KUKA KRL program: EPS_2_26115_ST7264_A_20260223020928.src

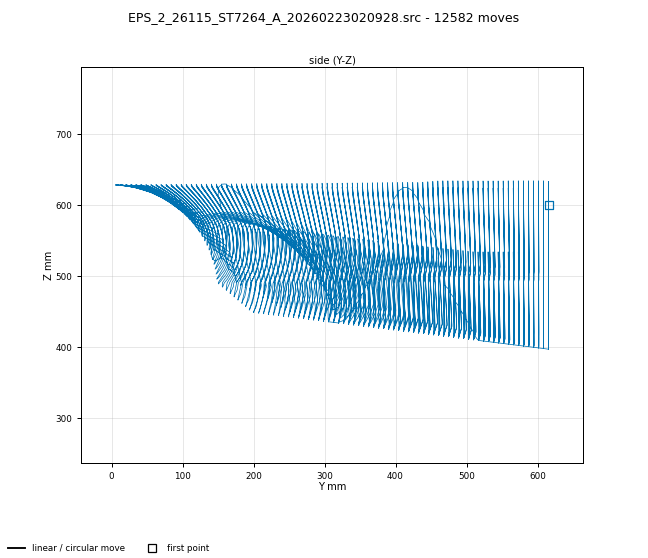
[picture p0: tool path of EPS_2_26115_ST7264_A_20260223020928.src, 12582 of 12584 moves have a stored position in this frame; points joined in program order, loops and branches not executed]
&ACCESS RVP
&REL 4
&COMMENT QRS 19112012
&PARAM EDITMASK = *
DEF PART()
EXT BAS (BAS_COMMAND :IN,REAL :IN )
INT I
BAS (#INITMOV,0 )

;KUKA QRS Post kuka4.cps  Date:22-06-2017 !

File_ID=3073

QRS_PRE_INIT()

;Init var - Until changes are made in qrs_pre_init
Outlet_Square_prg=0
Inlet_1_Square_prg=0
Inlet_2_Square_prg=0
Inlet_3_Square_prg=0
Inlet_4_Square_prg=0
Inlet_5_Square_prg=0

Outlet_1={X 0.000, Y 460.000, Z 509.000, B 0.000, E1 0.000 }
Inlet_1={X 0.000, Y 510.210, Z 499.000, B 0.000, E1 180.000 }
Inlet_2={X 0.000, Y 509.920, Z 385.000, B 0.000, E1 270.000 }
Outlet_1_type=251
Inlet_1_type=251
Inlet_2_type=299
;QRS#1=Sidecore dimensions
;QRS#2=250-10" PVC SDR 35 Cut Back
;QRS#3=250-10" PVC SDR 35
;QRS#4=300-12" PVC SDR 35
;QRS#5=
;QRS#6=
;QRS#7=
;QRS#8=
;QRS#9=14M PSX
;QRS#10=14M PSX
;QRS#11=16M PSX
;QRS#12=
;QRS#13=
;QRS#14=
;QRS#15=
;QRS#16=1220x127x914 3'
;QRS#17=EPS Height
;QRS#18=634,5
;QRS#19=*
;QRS#20= UPDATED VERSION 22-06-2017
;QRS#21=*
Outlet_Square=0100
Inlet_1_Square=0100
Inlet_2_Square=0150
Inlet_3_Square=0
Inlet_4_Square=0
Inlet_5_Square=0
Mill_Square=1
Outlet_Square_Prg=215
Inlet_1_Square_prg=205
Inlet_2_Square_prg=206

QRS_INIT()

$ADVANCE=5

; T1
PTP {E1 173.607,E2 173.607}
PTP {X 0,Y 615.507,A -85,B 0,C 180,E1 173.607,E2 173.607,E3 0,E4 0,E5 0,E6 0}
QRS_SPEED_INIT()
LIN {X 0,Y 615.507,Z 600,A -85,B 0,C 180,E1 173.607,E2 173.607,E3 0,E4 0,E5 0,E6 0} C_VEL
LIN {X 0,Y 615.507,Z 407.495,A -85,B 0,C 180,E1 173.607,E2 173.607} C_VEL
LIN {X 0,Y 615.507,Z 399.316,A -85,B 0,C 180,E1 173.607,E2 173.607} C_VEL
LIN {X 0,Y 615.491,Z 397.316,A -85,B 0,C 180,E1 173.42,E2 173.42} C_VEL
LIN {X 0,Y 615.489,Z 397.323,A -85,B 0,C 180,E1 170.801,E2 170.801} C_VEL
LIN {X 0,Y 615.489,Z 397.323,A -85,B 0,C 180,E1 168.139,E2 168.139} C_VEL
LIN {X 0,Y 615.493,Z 397.316,A -85,B 0,C 180,E1 165.451,E2 165.451} C_VEL
LIN {X 0,Y 615.49,Z 397.315,A -85,B 0,C 180,E1 162.729,E2 162.729} C_VEL
LIN {X 0,Y 615.484,Z 397.318,A -85,B 0,C 180,E1 159.967,E2 159.967} C_VEL
LIN {X 0,Y 615.477,Z 397.323,A -85,B 0,C 180,E1 157.155,E2 157.155} C_VEL
LIN {X 0,Y 615.499,Z 397.325,A -85,B 0,C 180,E1 154.429,E2 154.429} C_VEL
LIN {X 0,Y 615.497,Z 397.322,A -85,B 0,C 180,E1 151.548,E2 151.548} C_VEL
LIN {X 0,Y 615.483,Z 397.318,A -85,B 0,C 180,E1 148.915,E2 148.915} C_VEL
LIN {X 0,Y 615.484,Z 397.319,A -85,B 0,C 180,E1 146.466,E2 146.466} C_VEL
LIN {X 0,Y 615.488,Z 397.32,A -85,B 0,C 180,E1 143.575,E2 143.575} C_VEL
LIN {X 0,Y 615.496,Z 397.324,A -85,B 0,C 180,E1 140.937,E2 140.937} C_VEL
LIN {X 0,Y 615.485,Z 397.317,A -85,B 0,C 180,E1 138.526,E2 138.526} C_VEL
LIN {X 0,Y 615.495,Z 397.315,A -85,B 0,C 180,E1 135.851,E2 135.851} C_VEL
LIN {X 0,Y 615.485,Z 397.321,A -85,B 0,C 180,E1 133.047,E2 133.047} C_VEL
LIN {X 0,Y 615.492,Z 397.32,A -85,B 0,C 180,E1 130.089,E2 130.089} C_VEL
LIN {X 0,Y 615.497,Z 397.512,A -85,B 0,C 180,E1 127.721,E2 127.721} C_VEL
LIN {X 0,Y 615.499,Z 409.44,A -85,B 0,C 180,E1 124.814,E2 124.814} C_VEL
LIN {X 0,Y 615.489,Z 415.54,A -85,B 0,C 180,E1 123.236,E2 123.236} C_VEL
LIN {X 0,Y 615.477,Z 425.47,A -85,B 0,C 180,E1 120.54,E2 120.54} C_VEL
LIN {X 0,Y 615.485,Z 435.39,A -85,B 0,C 180,E1 117.915,E2 117.915} C_VEL
LIN {X 0,Y 615.488,Z 446.726,A -85,B 0,C 180,E1 114.992,E2 114.992} C_VEL
LIN {X 0,Y 615.49,Z 458.047,A -85,B 0,C 180,E1 112.136,E2 112.136} C_VEL
LIN {X 0,Y 615.483,Z 469.366,A -85,B 0,C 180,E1 109.338,E2 109.338} C_VEL
LIN {X 0,Y 615.48,Z 480.679,A -85,B 0,C 180,E1 106.587,E2 106.587} C_VEL
LIN {X 0,Y 615.493,Z 491.397,A -85,B 0,C 180,E1 104.013,E2 104.013} C_VEL
LIN {X 0,Y 615.494,Z 505.428,A -85,B 0,C 180,E1 103.79,E2 103.79} C_VEL
LIN {X 0,Y 615.479,Z 518.818,A -85,B 0,C 180,E1 103.454,E2 103.454} C_VEL
LIN {X 0,Y 615.493,Z 532.069,A -85,B 0,C 180,E1 102.991,E2 102.991} C_VEL
LIN {X 0,Y 615.477,Z 545.74,A -85,B 0,C 180,E1 102.363,E2 102.363} C_VEL
LIN {X 0,Y 615.499,Z 557.359,A -85,B 0,C 180,E1 101.694,E2 101.694} C_VEL
LIN {X 0,Y 615.496,Z 568.763,A -85,B 0,C 180,E1 100.891,E2 100.891} C_VEL
LIN {X 0,Y 615.498,Z 578.93,A -85,B 0,C 180,E1 100.028,E2 100.028} C_VEL
LIN {X 0,Y 615.497,Z 588.665,A -85,B 0,C 180,E1 99.033,E2 99.033} C_VEL
LIN {X 0,Y 615.498,Z 596.737,A -85,B 0,C 180,E1 98.041,E2 98.041} C_VEL
LIN {X 0,Y 615.494,Z 604.38,A -85,B 0,C 180,E1 96.899,E2 96.899} C_VEL
LIN {X 0,Y 615.497,Z 609.85,A -85,B 0,C 180,E1 95.898,E2 95.898} C_VEL
LIN {X 0,Y 615.494,Z 615.515,A -85,B 0,C 180,E1 94.585,E2 94.585} C_VEL
LIN {X 0,Y 615.494,Z 619.633,A -85,B 0,C 180,E1 93.273,E2 93.273} C_VEL
LIN {X 0,Y 615.499,Z 622.33,A -85,B 0,C 180,E1 91.963,E2 91.963} C_VEL
LIN {X 0,Y 615.491,Z 623.692,A -85,B 0,C 180,E1 90.654,E2 90.654} C_VEL
LIN {X 0,Y 615.492,Z 623.747,A -85,B 0,C 180,E1 89.346,E2 89.346} C_VEL
LIN {X 0,Y 615.499,Z 622.481,A -85,B 0,C 180,E1 88.037,E2 88.037} C_VEL
LIN {X 0,Y 615.494,Z 619.875,A -85,B 0,C 180,E1 86.727,E2 86.727} C_VEL
LIN {X 0,Y 615.495,Z 615.851,A -85,B 0,C 180,E1 85.416,E2 85.416} C_VEL
LIN {X 0,Y 615.498,Z 610.289,A -85,B 0,C 180,E1 84.102,E2 84.102} C_VEL
LIN {X 0,Y 615.495,Z 604.933,A -85,B 0,C 180,E1 83.102,E2 83.102} C_VEL
LIN {X 0,Y 615.498,Z 597.407,A -85,B 0,C 180,E1 81.959,E2 81.959} C_VEL
LIN {X 0,Y 615.496,Z 589.471,A -85,B 0,C 180,E1 80.967,E2 80.967} C_VEL
LIN {X 0,Y 615.496,Z 579.888,A -85,B 0,C 180,E1 79.972,E2 79.972} C_VEL
LIN {X 0,Y 615.497,Z 569.893,A -85,B 0,C 180,E1 79.108,E2 79.108} C_VEL
LIN {X 0,Y 615.5,Z 558.732,A -85,B 0,C 180,E1 78.306,E2 78.306} C_VEL
LIN {X 0,Y 615.48,Z 547.42,A -85,B 0,C 180,E1 77.637,E2 77.637} C_VEL
LIN {X 0,Y 615.497,Z 535.177,A -85,B 0,C 180,E1 77.051,E2 77.051} C_VEL
LIN {X 0,Y 615.48,Z 521.631,A -85,B 0,C 180,E1 76.546,E2 76.546} C_VEL
LIN {X 0,Y 615.498,Z 507.581,A -85,B 0,C 180,E1 76.168,E2 76.168} C_VEL
LIN {X 0,Y 615.489,Z 493.874,A -85,B 0,C 180,E1 75.93,E2 75.93} C_VEL
LIN {X 0,Y 615.485,Z 491.294,A -85,B 0,C 180,E1 75.872,E2 75.872} C_VEL
LIN {X 0,Y 615.491,Z 479.633,A -85,B 0,C 180,E1 73.072,E2 73.072} C_VEL
LIN {X 0,Y 615.489,Z 468.32,A -85,B 0,C 180,E1 70.315,E2 70.315} C_VEL
LIN {X 0,Y 615.487,Z 457.571,A -85,B 0,C 180,E1 67.655,E2 67.655} C_VEL
LIN {X 0,Y 615.488,Z 447.078,A -85,B 0,C 180,E1 65.008,E2 65.008} C_VEL
LIN {X 0,Y 615.485,Z 435.734,A -85,B 0,C 180,E1 62.085,E2 62.085} C_VEL
LIN {X 0,Y 615.477,Z 425.807,A -85,B 0,C 180,E1 59.46,E2 59.46} C_VEL
LIN {X 0,Y 615.492,Z 415.867,A -85,B 0,C 180,E1 56.764,E2 56.764} C_VEL
LIN {X 0,Y 615.499,Z 409.806,A -85,B 0,C 180,E1 55.186,E2 55.186} C_VEL
LIN {X 0,Y 615.496,Z 398.283,A -85,B 0,C 180,E1 52.375,E2 52.375} C_VEL
LIN {X 0,Y 615.492,Z 397.32,A -85,B 0,C 180,E1 52.085,E2 52.085} C_VEL
LIN {X 0,Y 615.482,Z 397.322,A -85,B 0,C 180,E1 49.393,E2 49.393} C_VEL
LIN {X 0,Y 615.482,Z 397.325,A -85,B 0,C 180,E1 46.755,E2 46.755} C_VEL
LIN {X 0,Y 615.486,Z 397.325,A -85,B 0,C 180,E1 43.997,E2 43.997} C_VEL
LIN {X 0,Y 615.487,Z 397.323,A -85,B 0,C 180,E1 41.474,E2 41.474} C_VEL
LIN {X 0,Y 615.476,Z 397.323,A -85,B 0,C 180,E1 38.905,E2 38.905} C_VEL
LIN {X 0,Y 615.493,Z 397.319,A -85,B 0,C 180,E1 36.425,E2 36.425} C_VEL
LIN {X 0,Y 615.486,Z 397.324,A -85,B 0,C 180,E1 33.534,E2 33.534} C_VEL
LIN {X 0,Y 615.494,Z 397.326,A -85,B 0,C 180,E1 30.919,E2 30.919} C_VEL
LIN {X 0,Y 615.497,Z 397.324,A -85,B 0,C 180,E1 28.452,E2 28.452} C_VEL
LIN {X 0,Y 615.485,Z 397.321,A -85,B 0,C 180,E1 25.568,E2 25.568} C_VEL
LIN {X 0,Y 615.481,Z 397.323,A -85,B 0,C 180,E1 22.845,E2 22.845} C_VEL
LIN {X 0,Y 615.488,Z 397.326,A -85,B 0,C 180,E1 20.033,E2 20.033} C_VEL
LIN {X 0,Y 615.49,Z 397.32,A -85,B 0,C 180,E1 17.271,E2 17.271} C_VEL
LIN {X 0,Y 615.478,Z 397.323,A -85,B 0,C 180,E1 16.037,E2 16.037} C_VEL
LIN {X 0,Y 615.485,Z 413.535,A -85,B 0,C 180,E1 15.608,E2 15.608} C_VEL
LIN {X 0,Y 615.487,Z 427.783,A -85,B 0,C 180,E1 15.099,E2 15.099} C_VEL
LIN {X 0,Y 615.496,Z 441.504,A -85,B 0,C 180,E1 14.472,E2 14.472} C_VEL
LIN {X 0,Y 615.496,Z 455.075,A -85,B 0,C 180,E1 13.706,E2 13.706} C_VEL
LIN {X 0,Y 615.496,Z 468.458,A -85,B 0,C 180,E1 12.781,E2 12.781} C_VEL
LIN {X 0,Y 615.495,Z 479.572,A -85,B 0,C 180,E1 11.861,E2 11.861} C_VEL
LIN {X 0,Y 615.493,Z 489.483,A -85,B 0,C 180,E1 10.89,E2 10.89} C_VEL
LIN {X 0,Y 615.494,Z 499.761,A -85,B 0,C 180,E1 9.696,E2 9.696} C_VEL
LIN {X 0,Y 615.496,Z 508.028,A -85,B 0,C 180,E1 8.537,E2 8.537} C_VEL
LIN {X 0,Y 615.493,Z 515.783,A -85,B 0,C 180,E1 7.216,E2 7.216} C_VEL
LIN {X 0,Y 615.489,Z 521.95,A -85,B 0,C 180,E1 5.899,E2 5.899} C_VEL
LIN {X 0,Y 615.494,Z 526.715,A -85,B 0,C 180,E1 4.585,E2 4.585} C_VEL
LIN {X 0,Y 615.495,Z 530.22,A -85,B 0,C 180,E1 3.273,E2 3.273} C_VEL
LIN {X 0,Y 615.493,Z 532.541,A -85,B 0,C 180,E1 1.963,E2 1.963} C_VEL
LIN {X 0,Y 615.489,Z 533.728,A -85,B 0,C 180,E1 0.654,E2 0.654} C_VEL
LIN {X 0,Y 615.493,Z 533.751,A -85,B 0,C 180,E1 -0.654,E2 -0.654} C_VEL
LIN {X 0,Y 615.496,Z 532.646,A -85,B 0,C 180,E1 -1.963,E2 -1.963} C_VEL
LIN {X 0,Y 615.498,Z 530.415,A -85,B 0,C 180,E1 -3.273,E2 -3.273} C_VEL
LIN {X 0,Y 615.49,Z 527.005,A -85,B 0,C 180,E1 -4.584,E2 -4.584} C_VEL
LIN {X 0,Y 615.49,Z 522.337,A -85,B 0,C 180,E1 -5.898,E2 -5.898} C_VEL
LIN {X 0,Y 615.492,Z 516.272,A -85,B 0,C 180,E1 -7.216,E2 -7.216} C_VEL
LIN {X 0,Y 615.493,Z 508.633,A -85,B 0,C 180,E1 -8.537,E2 -8.537} C_VEL
LIN {X 0,Y 615.496,Z 500.45,A -85,B 0,C 180,E1 -9.696,E2 -9.696} C_VEL
LIN {X 0,Y 615.496,Z 490.332,A -85,B 0,C 180,E1 -10.891,E2 -10.891} C_VEL
LIN {X 0,Y 615.497,Z 478.683,A -85,B 0,C 180,E1 -12.028,E2 -12.028} C_VEL
LIN {X 0,Y 615.498,Z 467.412,A -85,B 0,C 180,E1 -12.949,E2 -12.949} C_VEL
LIN {X 0,Y 615.498,Z 455.173,A -85,B 0,C 180,E1 -13.79,E2 -13.79} C_VEL
LIN {X 0,Y 615.49,Z 441.774,A -85,B 0,C 180,E1 -14.549,E2 -14.549} C_VEL
LIN {X 0,Y 615.484,Z 427.91,A -85,B 0,C 180,E1 -15.184,E2 -15.184} C_VEL
LIN {X 0,Y 615.488,Z 413.693,A -85,B 0,C 180,E1 -15.693,E2 -15.693} C_VEL
LIN {X 0,Y 615.493,Z 399.614,A -85,B 0,C 180,E1 -16.07,E2 -16.07} C_VEL
LIN {X 0,Y 615.493,Z 397.326,A -85,B 0,C 180,E1 -16.135,E2 -16.135} C_VEL
LIN {X 0,Y 615.483,Z 397.313,A -85,B 0,C 180,E1 -18.646,E2 -18.646} C_VEL
LIN {X 0,Y 615.496,Z 397.309,A -85,B 0,C 180,E1 -21.432,E2 -21.432} C_VEL
LIN {X 0,Y 615.49,Z 397.317,A -85,B 0,C 180,E1 -24.272,E2 -24.272} C_VEL
LIN {X 0,Y 615.477,Z 397.311,A -85,B 0,C 180,E1 -27.043,E2 -27.043} C_VEL
LIN {X 0,Y 615.498,Z 397.324,A -85,B 0,C 180,E1 -29.796,E2 -29.796} C_VEL
LIN {X 0,Y 615.489,Z 397.309,A -85,B 0,C 180,E1 -32.457,E2 -32.457} C_VEL
LIN {X 0,Y 615.477,Z 397.31,A -85,B 0,C 180,E1 -34.816,E2 -34.816} C_VEL
LIN {X 0,Y 615.491,Z 397.314,A -85,B 0,C 180,E1 -37.242,E2 -37.242} C_VEL
LIN {X 0,Y 615.487,Z 397.313,A -85,B 0,C 180,E1 -40.089,E2 -40.089} C_VEL
LIN {X 0,Y 615.493,Z 397.307,A -85,B 0,C 180,E1 -42.353,E2 -42.353} C_VEL
LIN {X 0,Y 615.481,Z 397.38,A -85,B 0,C 180,E1 -45.035,E2 -45.035} C_VEL
LIN {X 0,Y 615.495,Z 409.15,A -85,B 0,C 180,E1 -47.648,E2 -47.648} C_VEL
LIN {X 0,Y 615.492,Z 411.649,A -85,B 0,C 180,E1 -48.224,E2 -48.224} C_VEL
LIN {X 0,Y 615.493,Z 419.889,A -85,B 0,C 180,E1 -51.096,E2 -51.096} C_VEL
LIN {X 0,Y 615.479,Z 427.226,A -85,B 0,C 180,E1 -53.575,E2 -53.575} C_VEL
LIN {X 0,Y 615.482,Z 434.558,A -85,B 0,C 180,E1 -55.978,E2 -55.978} C_VEL
LIN {X 0,Y 615.487,Z 441.885,A -85,B 0,C 180,E1 -58.314,E2 -58.314} C_VEL
LIN {X 0,Y 615.486,Z 450.435,A -85,B 0,C 180,E1 -60.968,E2 -60.968} C_VEL
LIN {X 0,Y 615.482,Z 458.971,A -85,B 0,C 180,E1 -63.556,E2 -63.556} C_VEL
LIN {X 0,Y 615.482,Z 467.193,A -85,B 0,C 180,E1 -65.993,E2 -65.993} C_VEL
LIN {X 0,Y 615.492,Z 477.256,A -85,B 0,C 180,E1 -68.919,E2 -68.919} C_VEL
LIN {X 0,Y 615.478,Z 487.085,A -85,B 0,C 180,E1 -71.72,E2 -71.72} C_VEL
LIN {X 0,Y 615.487,Z 496.738,A -85,B 0,C 180,E1 -74.435,E2 -74.435} C_VEL
LIN {X 0,Y 615.49,Z 502.185,A -85,B 0,C 180,E1 -75.949,E2 -75.949} C_VEL
LIN {X 0,Y 615.49,Z 517.456,A -85,B 0,C 180,E1 -76.21,E2 -76.21} C_VEL
LIN {X 0,Y 615.483,Z 531.54,A -85,B 0,C 180,E1 -76.589,E2 -76.589} C_VEL
LIN {X 0,Y 615.497,Z 544.122,A -85,B 0,C 180,E1 -77.051,E2 -77.051} C_VEL
LIN {X 0,Y 615.479,Z 556.579,A -85,B 0,C 180,E1 -77.637,E2 -77.637} C_VEL
LIN {X 0,Y 615.498,Z 569.319,A -85,B 0,C 180,E1 -78.39,E2 -78.39} C_VEL
LIN {X 0,Y 615.498,Z 580.481,A -85,B 0,C 180,E1 -79.2,E2 -79.2} C_VEL
LIN {X 0,Y 615.498,Z 591.177,A -85,B 0,C 180,E1 -80.138,E2 -80.138} C_VEL
LIN {X 0,Y 615.498,Z 600.542,A -85,B 0,C 180,E1 -81.133,E2 -81.133} C_VEL
LIN {X 0,Y 615.494,Z 608.303,A -85,B 0,C 180,E1 -82.124,E2 -82.124} C_VEL
LIN {X 0,Y 615.495,Z 614.653,A -85,B 0,C 180,E1 -83.101,E2 -83.101} C_VEL
LIN {X 0,Y 615.494,Z 620.07,A -85,B 0,C 180,E1 -84.102,E2 -84.102} C_VEL
LIN {X 0,Y 615.495,Z 625.683,A -85,B 0,C 180,E1 -85.416,E2 -85.416} C_VEL
LIN {X 0,Y 615.495,Z 629.754,A -85,B 0,C 180,E1 -86.727,E2 -86.727} C_VEL
LIN {X 0,Y 615.497,Z 632.406,A -85,B 0,C 180,E1 -88.037,E2 -88.037} C_VEL
LIN {X 0,Y 615.493,Z 633.723,A -85,B 0,C 180,E1 -89.346,E2 -89.346} C_VEL
LIN {X 0,Y 615.493,Z 633.723,A -85,B 0,C 180,E1 -90.654,E2 -90.654} C_VEL
LIN {X 0,Y 615.497,Z 632.406,A -85,B 0,C 180,E1 -91.963,E2 -91.963} C_VEL
LIN {X 0,Y 615.495,Z 629.754,A -85,B 0,C 180,E1 -93.273,E2 -93.273} C_VEL
LIN {X 0,Y 615.495,Z 625.683,A -85,B 0,C 180,E1 -94.585,E2 -94.585} C_VEL
LIN {X 0,Y 615.494,Z 620.07,A -85,B 0,C 180,E1 -95.898,E2 -95.898} C_VEL
LIN {X 0,Y 615.495,Z 614.653,A -85,B 0,C 180,E1 -96.899,E2 -96.899} C_VEL
LIN {X 0,Y 615.496,Z 607.072,A -85,B 0,C 180,E1 -98.041,E2 -98.041} C_VEL
LIN {X 0,Y 615.498,Z 597.587,A -85,B 0,C 180,E1 -99.199,E2 -99.199} C_VEL
LIN {X 0,Y 615.498,Z 587.641,A -85,B 0,C 180,E1 -100.194,E2 -100.194} C_VEL
LIN {X 0,Y 615.498,Z 576.384,A -85,B 0,C 180,E1 -101.118,E2 -101.118} C_VEL
LIN {X 0,Y 615.496,Z 565.414,A -85,B 0,C 180,E1 -101.861,E2 -101.861} C_VEL
LIN {X 0,Y 615.479,Z 553.329,A -85,B 0,C 180,E1 -102.53,E2 -102.53} C_VEL
LIN {X 0,Y 615.487,Z 539.928,A -85,B 0,C 180,E1 -103.117,E2 -103.117} C_VEL
LIN {X 0,Y 615.486,Z 525.894,A -85,B 0,C 180,E1 -103.58,E2 -103.58} C_VEL
LIN {X 0,Y 615.496,Z 511.623,A -85,B 0,C 180,E1 -103.905,E2 -103.905} C_VEL
LIN {X 0,Y 615.49,Z 502.185,A -85,B 0,C 180,E1 -104.051,E2 -104.051} C_VEL
LIN {X 0,Y 615.493,Z 491.87,A -85,B 0,C 180,E1 -106.928,E2 -106.928} C_VEL
LIN {X 0,Y 615.485,Z 482.134,A -85,B 0,C 180,E1 -109.685,E2 -109.685} C_VEL
LIN {X 0,Y 615.477,Z 472.891,A -85,B 0,C 180,E1 -112.343,E2 -112.343} C_VEL
LIN {X 0,Y 615.488,Z 463.851,A -85,B 0,C 180,E1 -114.992,E2 -114.992} C_VEL
LIN {X 0,Y 615.485,Z 454.091,A -85,B 0,C 180,E1 -117.915,E2 -117.915} C_VEL
LIN {X 0,Y 615.487,Z 445.55,A -85,B 0,C 180,E1 -120.539,E2 -120.539} C_VEL
LIN {X 0,Y 615.479,Z 437,A -85,B 0,C 180,E1 -123.237,E2 -123.237} C_VEL
LIN {X 0,Y 615.49,Z 429.008,A -85,B 0,C 180,E1 -125.834,E2 -125.834} C_VEL
LIN {X 0,Y 615.481,Z 421.113,A -85,B 0,C 180,E1 -128.486,E2 -128.486} C_VEL
LIN {X 0,Y 615.489,Z 413.616,A -85,B 0,C 180,E1 -131.095,E2 -131.095} C_VEL
LIN {X 0,Y 615.493,Z 406.106,A -85,B 0,C 180,E1 -133.619,E2 -133.619} C_VEL
LIN {X 0,Y 615.495,Z 398.096,A -85,B 0,C 180,E1 -136.381,E2 -136.381} C_VEL
LIN {X 0,Y 615.497,Z 397.316,A -85,B 0,C 180,E1 -136.756,E2 -136.756} C_VEL
LIN {X 0,Y 615.485,Z 397.328,A -85,B 0,C 180,E1 -139.393,E2 -139.393} C_VEL
LIN {X 0,Y 615.482,Z 397.32,A -85,B 0,C 180,E1 -141.989,E2 -141.989} C_VEL
LIN {X 0,Y 615.485,Z 397.318,A -85,B 0,C 180,E1 -144.384,E2 -144.384} C_VEL
LIN {X 0,Y 615.491,Z 397.323,A -85,B 0,C 180,E1 -146.764,E2 -146.764} C_VEL
LIN {X 0,Y 615.478,Z 397.318,A -85,B 0,C 180,E1 -149.08,E2 -149.08} C_VEL
LIN {X 0,Y 615.497,Z 397.322,A -85,B 0,C 180,E1 -151.548,E2 -151.548} C_VEL
LIN {X 0,Y 615.498,Z 397.325,A -85,B 0,C 180,E1 -154.429,E2 -154.429} C_VEL
LIN {X 0,Y 615.486,Z 397.321,A -85,B 0,C 180,E1 -157.155,E2 -157.155} C_VEL
LIN {X 0,Y 615.481,Z 397.319,A -85,B 0,C 180,E1 -159.967,E2 -159.967} C_VEL
LIN {X 0,Y 615.491,Z 397.315,A -85,B 0,C 180,E1 -162.73,E2 -162.73} C_VEL
LIN {X 0,Y 615.49,Z 397.317,A -85,B 0,C 180,E1 -165.451,E2 -165.451} C_VEL
LIN {X 0,Y 615.491,Z 397.322,A -85,B 0,C 180,E1 -168.139,E2 -168.139} C_VEL
LIN {X 0,Y 615.494,Z 397.322,A -85,B 0,C 180,E1 -170.801,E2 -170.801} C_VEL
LIN {X 0,Y 615.492,Z 397.316,A -85,B 0,C 180,E1 -173.443,E2 -173.443} C_VEL
LIN {X 0,Y 615.476,Z 397.319,A -85,B 0,C 180,E1 -176.071,E2 -176.071} C_VEL
LIN {X 0,Y 615.485,Z 397.323,A -85,B 0,C 180,E1 -178.691,E2 -178.691} C_VEL
LIN {X 0,Y 615.486,Z 397.323,A -85,B 0,C 180,E1 -181.309,E2 -181.309} C_VEL
LIN {X 0,Y 615.476,Z 397.319,A -85,B 0,C 180,E1 -183.929,E2 -183.929} C_VEL
LIN {X 0,Y 615.491,Z 397.316,A -85,B 0,C 180,E1 -186.58,E2 -186.58} C_VEL
LIN {X 0,Y 614.811,Z 397.468,A -85,B 0,C 180,E1 -187.126,E2 -187.126} C_VEL
LIN {X 0,Y 611.977,Z 397.879,A -85,B 0,C 180,E1 -188.012,E2 -188.012} C_VEL
LIN {X 0,Y 609.587,Z 398.19,A -85,B 0,C 180,E1 -188.724,E2 -188.724} C_VEL
LIN {X 0,Y 608.55,Z 398.308,A -85,B 0,C 180,E1 -189.274,E2 -189.274} C_VEL
LIN {X 0,Y 608.459,Z 398.317,A -85,B 0,C 180,E1 -189.46,E2 -189.46} C_VEL
LIN {X 0,Y 608.464,Z 398.321,A -85,B 0,C 180,E1 -192,E2 -192} C_VEL
LIN {X 0,Y 608.482,Z 398.315,A -85,B 0,C 180,E1 -194.72,E2 -194.72} C_VEL
LIN {X 0,Y 608.454,Z 398.317,A -85,B 0,C 180,E1 -197.477,E2 -197.477} C_VEL
LIN {X 0,Y 608.464,Z 398.316,A -85,B 0,C 180,E1 -200.274,E2 -200.274} C_VEL
LIN {X 0,Y 608.461,Z 398.321,A -85,B 0,C 180,E1 -202.476,E2 -202.476} C_VEL
LIN {X 0,Y 608.455,Z 398.317,A -85,B 0,C 180,E1 -204.571,E2 -204.571} C_VEL
LIN {X 0,Y 608.488,Z 398.317,A -85,B 0,C 180,E1 -207.209,E2 -207.209} C_VEL
LIN {X 0,Y 608.465,Z 398.32,A -85,B 0,C 180,E1 -209.971,E2 -209.971} C_VEL
LIN {X 0,Y 608.464,Z 398.319,A -85,B 0,C 180,E1 -212.879,E2 -212.879} C_VEL
LIN {X 0,Y 608.437,Z 398.319,A -85,B 0,C 180,E1 -215.278,E2 -215.278} C_VEL
LIN {X 0,Y 608.473,Z 398.319,A -85,B 0,C 180,E1 -217.746,E2 -217.746} C_VEL
LIN {X 0,Y 608.453,Z 398.319,A -85,B 0,C 180,E1 -220.329,E2 -220.329} C_VEL
LIN {X 0,Y 608.452,Z 398.317,A -85,B 0,C 180,E1 -222.96,E2 -222.96} C_VEL
LIN {X 0,Y 608.45,Z 398.318,A -85,B 0,C 180,E1 -225.737,E2 -225.737} C_VEL
LIN {X 0,Y 608.457,Z 398.317,A -85,B 0,C 180,E1 -228.659,E2 -228.659} C_VEL
LIN {X 0,Y 608.471,Z 398.318,A -85,B 0,C 180,E1 -231.412,E2 -231.412} C_VEL
LIN {X 0,Y 608.501,Z 398.517,A -85,B 0,C 180,E1 -232.195,E2 -232.195} C_VEL
LIN {X 0,Y 608.517,Z 410.265,A -85,B 0,C 180,E1 -235.086,E2 -235.086} C_VEL
LIN {X 0,Y 608.534,Z 418.387,A -85,B 0,C 180,E1 -237.125,E2 -237.125} C_VEL
LIN {X 0,Y 608.519,Z 428.094,A -85,B 0,C 180,E1 -239.779,E2 -239.779} C_VEL
LIN {X 0,Y 608.518,Z 439.411,A -85,B 0,C 180,E1 -242.786,E2 -242.786} C_VEL
LIN {X 0,Y 608.492,Z 449.626,A -85,B 0,C 180,E1 -245.431,E2 -245.431} C_VEL
LIN {X 0,Y 608.48,Z 460.986,A -85,B 0,C 180,E1 -248.309,E2 -248.309} C_VEL
LIN {X 0,Y 608.47,Z 472.973,A -85,B 0,C 180,E1 -251.285,E2 -251.285} C_VEL
LIN {X 0,Y 608.448,Z 483.708,A -85,B 0,C 180,E1 -253.906,E2 -253.906} C_VEL
LIN {X 0,Y 608.464,Z 491.868,A -85,B 0,C 180,E1 -255.828,E2 -255.828} C_VEL
LIN {X 0,Y 608.608,Z 506.72,A -85,B 0,C 180,E1 -256.079,E2 -256.079} C_VEL
LIN {X 0,Y 608.572,Z 520.189,A -85,B 0,C 180,E1 -256.433,E2 -256.433} C_VEL
LIN {X 0,Y 608.569,Z 533.115,A -85,B 0,C 180,E1 -256.901,E2 -256.901} C_VEL
LIN {X 0,Y 608.522,Z 545.809,A -85,B 0,C 180,E1 -257.494,E2 -257.494} C_VEL
LIN {X 0,Y 608.531,Z 558.745,A -85,B 0,C 180,E1 -258.255,E2 -258.255} C_VEL
LIN {X 0,Y 608.488,Z 570.554,A -85,B 0,C 180,E1 -259.112,E2 -259.112} C_VEL
LIN {X 0,Y 608.473,Z 580.915,A -85,B 0,C 180,E1 -260.023,E2 -260.023} C_VEL
LIN {X 0,Y 608.472,Z 590.427,A -85,B 0,C 180,E1 -261.029,E2 -261.029} C_VEL
LIN {X 0,Y 608.454,Z 599.496,A -85,B 0,C 180,E1 -262.2,E2 -262.2} C_VEL
LIN {X 0,Y 608.446,Z 606.967,A -85,B 0,C 180,E1 -263.397,E2 -263.397} C_VEL
LIN {X 0,Y 608.436,Z 613.376,A -85,B 0,C 180,E1 -264.698,E2 -264.698} C_VEL
LIN {X 0,Y 608.434,Z 618.298,A -85,B 0,C 180,E1 -266.026,E2 -266.026} C_VEL
LIN {X 0,Y 608.425,Z 621.734,A -85,B 0,C 180,E1 -267.352,E2 -267.352} C_VEL
LIN {X 0,Y 608.446,Z 623.778,A -85,B 0,C 180,E1 -268.676,E2 -268.676} C_VEL
LIN {X 0,Y 608.434,Z 624.495,A -85,B 0,C 180,E1 -270,E2 -270} C_VEL
LIN {X 0,Y 608.443,Z 623.882,A -85,B 0,C 180,E1 -271.324,E2 -271.324} C_VEL
LIN {X 0,Y 608.421,Z 621.929,A -85,B 0,C 180,E1 -272.648,E2 -272.648} C_VEL
LIN {X 0,Y 608.434,Z 618.585,A -85,B 0,C 180,E1 -273.974,E2 -273.974} C_VEL
LIN {X 0,Y 608.44,Z 613.761,A -85,B 0,C 180,E1 -275.302,E2 -275.302} C_VEL
LIN {X 0,Y 608.443,Z 607.473,A -85,B 0,C 180,E1 -276.601,E2 -276.601} C_VEL
LIN {X 0,Y 608.454,Z 600.1,A -85,B 0,C 180,E1 -277.8,E2 -277.8} C_VEL
LIN {X 0,Y 608.476,Z 592.564,A -85,B 0,C 180,E1 -278.803,E2 -278.803} C_VEL
LIN {X 0,Y 608.486,Z 583.518,A -85,B 0,C 180,E1 -279.809,E2 -279.809} C_VEL
LIN {X 0,Y 608.507,Z 572.723,A -85,B 0,C 180,E1 -280.804,E2 -280.804} C_VEL
LIN {X 0,Y 608.523,Z 561.383,A -85,B 0,C 180,E1 -281.661,E2 -281.661} C_VEL
LIN {X 0,Y 608.53,Z 549.039,A -85,B 0,C 180,E1 -282.422,E2 -282.422} C_VEL
LIN {X 0,Y 608.557,Z 537.172,A -85,B 0,C 180,E1 -283.015,E2 -283.015} C_VEL
LIN {X 0,Y 608.564,Z 524.221,A -85,B 0,C 180,E1 -283.524,E2 -283.524} C_VEL
LIN {X 0,Y 608.594,Z 509.989,A -85,B 0,C 180,E1 -283.936,E2 -283.936} C_VEL
LIN {X 0,Y 608.606,Z 495.668,A -85,B 0,C 180,E1 -284.207,E2 -284.207} C_VEL
LIN {X 0,Y 608.45,Z 491.646,A -85,B 0,C 180,E1 -284.268,E2 -284.268} C_VEL
LIN {X 0,Y 608.482,Z 479.817,A -85,B 0,C 180,E1 -287.129,E2 -287.129} C_VEL
LIN {X 0,Y 608.459,Z 468.45,A -85,B 0,C 180,E1 -289.922,E2 -289.922} C_VEL
LIN {X 0,Y 608.485,Z 457.083,A -85,B 0,C 180,E1 -292.763,E2 -292.763} C_VEL
LIN {X 0,Y 608.513,Z 445.468,A -85,B 0,C 180,E1 -295.728,E2 -295.728} C_VEL
LIN {X 0,Y 608.521,Z 435.766,A -85,B 0,C 180,E1 -298.263,E2 -298.263} C_VEL
LIN {X 0,Y 608.551,Z 425.881,A -85,B 0,C 180,E1 -300.908,E2 -300.908} C_VEL
LIN {X 0,Y 608.514,Z 415.694,A -85,B 0,C 180,E1 -303.668,E2 -303.668} C_VEL
LIN {X 0,Y 608.524,Z 404.237,A -85,B 0,C 180,E1 -306.498,E2 -306.498} C_VEL
LIN {X 0,Y 608.459,Z 398.319,A -85,B 0,C 180,E1 -307.993,E2 -307.993} C_VEL
LIN {X 0,Y 608.446,Z 398.32,A -85,B 0,C 180,E1 -310.328,E2 -310.328} C_VEL
LIN {X 0,Y 608.45,Z 398.32,A -85,B 0,C 180,E1 -312.96,E2 -312.96} C_VEL
LIN {X 0,Y 608.463,Z 398.321,A -85,B 0,C 180,E1 -315.736,E2 -315.736} C_VEL
LIN {X 0,Y 608.463,Z 398.319,A -85,B 0,C 180,E1 -318.658,E2 -318.658} C_VEL
LIN {X 0,Y 608.47,Z 398.32,A -85,B 0,C 180,E1 -321.76,E2 -321.76} C_VEL
LIN {X 0,Y 608.481,Z 398.317,A -85,B 0,C 180,E1 -323.95,E2 -323.95} C_VEL
LIN {X 0,Y 608.451,Z 398.32,A -85,B 0,C 180,E1 -326.328,E2 -326.328} C_VEL
LIN {X 0,Y 608.464,Z 398.319,A -85,B 0,C 180,E1 -328.73,E2 -328.73} C_VEL
LIN {X 0,Y 608.477,Z 398.319,A -85,B 0,C 180,E1 -331.38,E2 -331.38} C_VEL
LIN {X 0,Y 608.445,Z 398.323,A -85,B 0,C 180,E1 -333.964,E2 -333.964} C_VEL
LIN {X 0,Y 608.472,Z 398.319,A -85,B 0,C 180,E1 -336.155,E2 -336.155} C_VEL
LIN {X 0,Y 608.471,Z 398.318,A -85,B 0,C 180,E1 -338.308,E2 -338.308} C_VEL
LIN {X 0,Y 608.477,Z 398.318,A -85,B 0,C 180,E1 -341.283,E2 -341.283} C_VEL
LIN {X 0,Y 608.465,Z 398.319,A -85,B 0,C 180,E1 -343.79,E2 -343.79} C_VEL
LIN {X 0,Y 608.666,Z 402.126,A -85,B 0,C 180,E1 -343.895,E2 -343.895} C_VEL
LIN {X 0,Y 608.643,Z 416.149,A -85,B 0,C 180,E1 -344.298,E2 -344.298} C_VEL
LIN {X 0,Y 608.613,Z 430.746,A -85,B 0,C 180,E1 -344.855,E2 -344.855} C_VEL
LIN {X 0,Y 608.569,Z 444.846,A -85,B 0,C 180,E1 -345.538,E2 -345.538} C_VEL
LIN {X 0,Y 608.554,Z 458.988,A -85,B 0,C 180,E1 -346.39,E2 -346.39} C_VEL
LIN {X 0,Y 608.528,Z 471.716,A -85,B 0,C 180,E1 -347.324,E2 -347.324} C_VEL
LIN {X 0,Y 608.497,Z 483.276,A -85,B 0,C 180,E1 -348.339,E2 -348.339} C_VEL
LIN {X 0,Y 608.476,Z 492.991,A -85,B 0,C 180,E1 -349.35,E2 -349.35} C_VEL
LIN {X 0,Y 608.477,Z 502.519,A -85,B 0,C 180,E1 -350.527,E2 -350.527} C_VEL
LIN {X 0,Y 608.457,Z 510.457,A -85,B 0,C 180,E1 -351.698,E2 -351.698} C_VEL
LIN {X 0,Y 608.44,Z 517.87,A -85,B 0,C 180,E1 -353.034,E2 -353.034} C_VEL
LIN {X 0,Y 608.447,Z 523.755,A -85,B 0,C 180,E1 -354.365,E2 -354.365} C_VEL
LIN {X 0,Y 608.429,Z 527.24,A -85,B 0,C 180,E1 -355.362,E2 -355.362} C_VEL
LIN {X 0,Y 608.423,Z 530.787,A -85,B 0,C 180,E1 -356.689,E2 -356.689} C_VEL
LIN {X 0,Y 608.438,Z 533.138,A -85,B 0,C 180,E1 -358.014,E2 -358.014} C_VEL
LIN {X 0,Y 608.432,Z 534.337,A -85,B 0,C 180,E1 -359.338,E2 -359.338} C_VEL
LIN {X 0,Y 608.436,Z 534.361,A -85,B 0,C 180,E1 -360.662,E2 -360.662} C_VEL
LIN {X 0,Y 608.442,Z 533.245,A -85,B 0,C 180,E1 -361.986,E2 -361.986} C_VEL
LIN {X 0,Y 608.426,Z 530.983,A -85,B 0,C 180,E1 -363.311,E2 -363.311} C_VEL
LIN {X 0,Y 608.425,Z 527.526,A -85,B 0,C 180,E1 -364.638,E2 -364.638} C_VEL
LIN {X 0,Y 608.431,Z 522.801,A -85,B 0,C 180,E1 -365.967,E2 -365.967} C_VEL
LIN {X 0,Y 608.457,Z 516.67,A -85,B 0,C 180,E1 -367.299,E2 -367.299} C_VEL
LIN {X 0,Y 608.468,Z 508.952,A -85,B 0,C 180,E1 -368.636,E2 -368.636} C_VEL
LIN {X 0,Y 608.471,Z 500.708,A -85,B 0,C 180,E1 -369.809,E2 -369.809} C_VEL
LIN {X 0,Y 608.478,Z 491.048,A -85,B 0,C 180,E1 -370.959,E2 -370.959} C_VEL
LIN {X 0,Y 608.509,Z 480.671,A -85,B 0,C 180,E1 -371.999,E2 -371.999} C_VEL
LIN {X 0,Y 608.533,Z 468.596,A -85,B 0,C 180,E1 -373.015,E2 -373.015} C_VEL
LIN {X 0,Y 608.564,Z 455.192,A -85,B 0,C 180,E1 -373.95,E2 -373.95} C_VEL
LIN {X 0,Y 608.59,Z 441.763,A -85,B 0,C 180,E1 -374.718,E2 -374.718} C_VEL
LIN {X 0,Y 608.615,Z 427.89,A -85,B 0,C 180,E1 -375.359,E2 -375.359} C_VEL
LIN {X 0,Y 608.646,Z 412.357,A -85,B 0,C 180,E1 -375.917,E2 -375.917} C_VEL
LIN {X 0,Y 608.483,Z 398.317,A -85,B 0,C 180,E1 -376.293,E2 -376.293} C_VEL
LIN {X 0,Y 608.456,Z 398.313,A -85,B 0,C 180,E1 -378.87,E2 -378.87} C_VEL
LIN {X 0,Y 608.476,Z 398.315,A -85,B 0,C 180,E1 -381.691,E2 -381.691} C_VEL
LIN {X 0,Y 608.452,Z 398.314,A -85,B 0,C 180,E1 -384.571,E2 -384.571} C_VEL
LIN {X 0,Y 608.475,Z 398.311,A -85,B 0,C 180,E1 -387.206,E2 -387.206} C_VEL
LIN {X 0,Y 608.475,Z 398.318,A -85,B 0,C 180,E1 -389.972,E2 -389.972} C_VEL
LIN {X 0,Y 608.464,Z 398.312,A -85,B 0,C 180,E1 -392.523,E2 -392.523} C_VEL
LIN {X 0,Y 608.445,Z 398.317,A -85,B 0,C 180,E1 -395.278,E2 -395.278} C_VEL
LIN {X 0,Y 608.47,Z 398.32,A -85,B 0,C 180,E1 -397.746,E2 -397.746} C_VEL
LIN {X 0,Y 608.449,Z 398.314,A -85,B 0,C 180,E1 -400.329,E2 -400.329} C_VEL
LIN {X 0,Y 608.484,Z 398.315,A -85,B 0,C 180,E1 -403.31,E2 -403.31} C_VEL
LIN {X 0,Y 608.453,Z 398.418,A -85,B 0,C 180,E1 -405.056,E2 -405.056} C_VEL
LIN {X 0,Y 608.458,Z 410.094,A -85,B 0,C 180,E1 -407.666,E2 -407.666} C_VEL
LIN {X 0,Y 608.543,Z 414.921,A -85,B 0,C 180,E1 -408.831,E2 -408.831} C_VEL
LIN {X 0,Y 608.537,Z 422.341,A -85,B 0,C 180,E1 -411.417,E2 -411.417} C_VEL
LIN {X 0,Y 608.522,Z 429.779,A -85,B 0,C 180,E1 -413.945,E2 -413.945} C_VEL
LIN {X 0,Y 608.509,Z 438.25,A -85,B 0,C 180,E1 -416.729,E2 -416.729} C_VEL
LIN {X 0,Y 608.511,Z 446.816,A -85,B 0,C 180,E1 -419.457,E2 -419.457} C_VEL
LIN {X 0,Y 608.497,Z 455.382,A -85,B 0,C 180,E1 -422.111,E2 -422.111} C_VEL
LIN {X 0,Y 608.461,Z 463.949,A -85,B 0,C 180,E1 -424.699,E2 -424.699} C_VEL
LIN {X 0,Y 608.461,Z 473.498,A -85,B 0,C 180,E1 -427.524,E2 -427.524} C_VEL
LIN {X 0,Y 608.452,Z 482.305,A -85,B 0,C 180,E1 -430.078,E2 -430.078} C_VEL
LIN {X 0,Y 608.454,Z 492.095,A -85,B 0,C 180,E1 -432.87,E2 -432.87} C_VEL
LIN {X 0,Y 608.436,Z 501.762,A -85,B 0,C 180,E1 -435.586,E2 -435.586} C_VEL
LIN {X 0,Y 608.457,Z 502.482,A -85,B 0,C 180,E1 -435.788,E2 -435.788} C_VEL
LIN {X 0,Y 608.588,Z 517.464,A -85,B 0,C 180,E1 -436.051,E2 -436.051} C_VEL
LIN {X 0,Y 608.576,Z 531.556,A -85,B 0,C 180,E1 -436.433,E2 -436.433} C_VEL
LIN {X 0,Y 608.57,Z 544.157,A -85,B 0,C 180,E1 -436.901,E2 -436.901} C_VEL
LIN {X 0,Y 608.523,Z 556.641,A -85,B 0,C 180,E1 -437.494,E2 -437.494} C_VEL
LIN {X 0,Y 608.531,Z 569.425,A -85,B 0,C 180,E1 -438.255,E2 -438.255} C_VEL
LIN {X 0,Y 608.499,Z 580.703,A -85,B 0,C 180,E1 -439.079,E2 -439.079} C_VEL
LIN {X 0,Y 608.472,Z 591.391,A -85,B 0,C 180,E1 -440.023,E2 -440.023} C_VEL
LIN {X 0,Y 608.473,Z 600.822,A -85,B 0,C 180,E1 -441.029,E2 -441.029} C_VEL
LIN {X 0,Y 608.453,Z 609.798,A -85,B 0,C 180,E1 -442.2,E2 -442.2} C_VEL
LIN {X 0,Y 608.442,Z 617.227,A -85,B 0,C 180,E1 -443.399,E2 -443.399} C_VEL
LIN {X 0,Y 608.44,Z 623.568,A -85,B 0,C 180,E1 -444.698,E2 -444.698} C_VEL
LIN {X 0,Y 608.431,Z 628.441,A -85,B 0,C 180,E1 -446.026,E2 -446.026} C_VEL
LIN {X 0,Y 608.424,Z 631.831,A -85,B 0,C 180,E1 -447.352,E2 -447.352} C_VEL
LIN {X 0,Y 608.442,Z 633.83,A -85,B 0,C 180,E1 -448.676,E2 -448.676} C_VEL
LIN {X 0,Y 608.433,Z 634.5,A -85,B 0,C 180,E1 -450,E2 -450} C_VEL
LIN {X 0,Y 608.442,Z 633.83,A -85,B 0,C 180,E1 -451.324,E2 -451.324} C_VEL
LIN {X 0,Y 608.424,Z 631.831,A -85,B 0,C 180,E1 -452.648,E2 -452.648} C_VEL
LIN {X 0,Y 608.431,Z 628.441,A -85,B 0,C 180,E1 -453.974,E2 -453.974} C_VEL
LIN {X 0,Y 608.44,Z 623.568,A -85,B 0,C 180,E1 -455.302,E2 -455.302} C_VEL
LIN {X 0,Y 608.445,Z 617.212,A -85,B 0,C 180,E1 -456.603,E2 -456.603} C_VEL
LIN {X 0,Y 608.453,Z 609.798,A -85,B 0,C 180,E1 -457.8,E2 -457.8} C_VEL
LIN {X 0,Y 608.473,Z 600.823,A -85,B 0,C 180,E1 -458.971,E2 -458.971} C_VEL
LIN {X 0,Y 608.472,Z 591.39,A -85,B 0,C 180,E1 -459.977,E2 -459.977} C_VEL
LIN {X 0,Y 608.506,Z 580.047,A -85,B 0,C 180,E1 -460.973,E2 -460.973} C_VEL
LIN {X 0,Y 608.534,Z 568.146,A -85,B 0,C 180,E1 -461.829,E2 -461.829} C_VEL
LIN {X 0,Y 608.517,Z 555.074,A -85,B 0,C 180,E1 -462.591,E2 -462.591} C_VEL
LIN {X 0,Y 608.552,Z 542.168,A -85,B 0,C 180,E1 -463.185,E2 -463.185} C_VEL
LIN {X 0,Y 608.588,Z 528.183,A -85,B 0,C 180,E1 -463.673,E2 -463.673} C_VEL
LIN {X 0,Y 608.622,Z 514.456,A -85,B 0,C 180,E1 -464.013,E2 -464.013} C_VEL
LIN {X 0,Y 608.459,Z 502.473,A -85,B 0,C 180,E1 -464.215,E2 -464.215} C_VEL
LIN {X 0,Y 608.451,Z 493.319,A -85,B 0,C 180,E1 -466.784,E2 -466.784} C_VEL
LIN {X 0,Y 608.459,Z 483.529,A -85,B 0,C 180,E1 -469.57,E2 -469.57} C_VEL
LIN {X 0,Y 608.461,Z 473.739,A -85,B 0,C 180,E1 -472.406,E2 -472.406} C_VEL
LIN {X 0,Y 608.474,Z 465.172,A -85,B 0,C 180,E1 -474.935,E2 -474.935} C_VEL
LIN {X 0,Y 608.472,Z 456.606,A -85,B 0,C 180,E1 -477.517,E2 -477.517} C_VEL
LIN {X 0,Y 608.5,Z 448.626,A -85,B 0,C 180,E1 -479.977,E2 -479.977} C_VEL
LIN {X 0,Y 608.525,Z 439.473,A -85,B 0,C 180,E1 -482.875,E2 -482.875} C_VEL
LIN {X 0,Y 608.535,Z 430.955,A -85,B 0,C 180,E1 -485.662,E2 -485.662} C_VEL
LIN {X 0,Y 608.533,Z 423.312,A -85,B 0,C 180,E1 -488.248,E2 -488.248} C_VEL
LIN {X 0,Y 608.558,Z 416.223,A -85,B 0,C 180,E1 -490.73,E2 -490.73} C_VEL
LIN {X 0,Y 608.521,Z 408.483,A -85,B 0,C 180,E1 -493.314,E2 -493.314} C_VEL
LIN {X 0,Y 608.568,Z 400.327,A -85,B 0,C 180,E1 -496.139,E2 -496.139} C_VEL
LIN {X 0,Y 608.472,Z 398.317,A -85,B 0,C 180,E1 -496.949,E2 -496.949} C_VEL
LIN {X 0,Y 608.454,Z 398.319,A -85,B 0,C 180,E1 -499.697,E2 -499.697} C_VEL
LIN {X 0,Y 608.469,Z 398.32,A -85,B 0,C 180,E1 -502.254,E2 -502.254} C_VEL
LIN {X 0,Y 608.443,Z 398.318,A -85,B 0,C 180,E1 -504.722,E2 -504.722} C_VEL
LIN {X 0,Y 608.465,Z 398.316,A -85,B 0,C 180,E1 -507.477,E2 -507.477} C_VEL
LIN {X 0,Y 608.469,Z 398.317,A -85,B 0,C 180,E1 -510.221,E2 -510.221} C_VEL
LIN {X 0,Y 608.487,Z 398.317,A -85,B 0,C 180,E1 -512.792,E2 -512.792} C_VEL
LIN {X 0,Y 608.455,Z 398.317,A -85,B 0,C 180,E1 -515.429,E2 -515.429} C_VEL
LIN {X 0,Y 608.471,Z 398.315,A -85,B 0,C 180,E1 -518.309,E2 -518.309} C_VEL
LIN {X 0,Y 608.471,Z 398.315,A -85,B 0,C 180,E1 -521.284,E2 -521.284} C_VEL
LIN {X 0,Y 608.458,Z 398.317,A -85,B 0,C 180,E1 -523.906,E2 -523.906} C_VEL
LIN {X 0,Y 608.461,Z 398.32,A -85,B 0,C 180,E1 -526.644,E2 -526.644} C_VEL
LIN {X 0,Y 608.467,Z 398.32,A -85,B 0,C 180,E1 -529.35,E2 -529.35} C_VEL
LIN {X 0,Y 608.471,Z 398.316,A -85,B 0,C 180,E1 -532.033,E2 -532.033} C_VEL
LIN {X 0,Y 608.465,Z 398.315,A -85,B 0,C 180,E1 -534.698,E2 -534.698} C_VEL
LIN {X 0,Y 608.482,Z 398.315,A -85,B 0,C 180,E1 -537.352,E2 -537.352} C_VEL
LIN {X 0,Y 608.477,Z 398.32,A -85,B 0,C 180,E1 -540,E2 -540} C_VEL
LIN {X 0,Y 608.485,Z 398.314,A -85,B 0,C 180,E1 -542.648,E2 -542.648} C_VEL
LIN {X 0,Y 608.464,Z 398.316,A -85,B 0,C 180,E1 -545.302,E2 -545.302} C_VEL
LIN {X 0,Y 608.475,Z 398.315,A -85,B 0,C 180,E1 -547.967,E2 -547.967} C_VEL
LIN {X 0,Y 608.459,Z 398.317,A -85,B 0,C 180,E1 -549.46,E2 -549.46} C_VEL
LIN {X 0,Y 607.776,Z 398.402,A -85,B 0,C 180,E1 -550.012,E2 -550.012} C_VEL
LIN {X 0,Y 604.924,Z 398.759,A -85,B 0,C 180,E1 -550.909,E2 -550.909} C_VEL
LIN {X 0,Y 602.525,Z 399.06,A -85,B 0,C 180,E1 -551.631,E2 -551.631} C_VEL
LIN {X 0,Y 601.495,Z 399.188,A -85,B 0,C 180,E1 -552.188,E2 -552.188} C_VEL
LIN {X 0,Y 601.411,Z 399.196,A -85,B 0,C 180,E1 -552.376,E2 -552.376} C_VEL
LIN {X 0,Y 601.435,Z 399.195,A -85,B 0,C 180,E1 -554.897,E2 -554.897} C_VEL
LIN {X 0,Y 601.434,Z 399.192,A -85,B 0,C 180,E1 -556.986,E2 -556.986} C_VEL
LIN {X 0,Y 601.408,Z 399.197,A -85,B 0,C 180,E1 -559.809,E2 -559.809} C_VEL
LIN {X 0,Y 601.418,Z 399.199,A -85,B 0,C 180,E1 -562.606,E2 -562.606} C_VEL
LIN {X 0,Y 601.404,Z 399.195,A -85,B 0,C 180,E1 -564.879,E2 -564.879} C_VEL
LIN {X 0,Y 601.422,Z 399.195,A -85,B 0,C 180,E1 -567.363,E2 -567.363} C_VEL
LIN {X 0,Y 601.43,Z 399.197,A -85,B 0,C 180,E1 -570.164,E2 -570.164} C_VEL
LIN {X 0,Y 601.428,Z 399.194,A -85,B 0,C 180,E1 -572.716,E2 -572.716} C_VEL
LIN {X 0,Y 601.392,Z 399.197,A -85,B 0,C 180,E1 -575.111,E2 -575.111} C_VEL
LIN {X 0,Y 601.437,Z 399.194,A -85,B 0,C 180,E1 -577.419,E2 -577.419} C_VEL
LIN {X 0,Y 601.404,Z 399.195,A -85,B 0,C 180,E1 -579.996,E2 -579.996} C_VEL
LIN {X 0,Y 601.415,Z 399.194,A -85,B 0,C 180,E1 -582.67,E2 -582.67} C_VEL
LIN {X 0,Y 601.429,Z 399.194,A -85,B 0,C 180,E1 -585.482,E2 -585.482} C_VEL
LIN {X 0,Y 601.422,Z 399.196,A -85,B 0,C 180,E1 -588.407,E2 -588.407} C_VEL
LIN {X 0,Y 601.438,Z 399.194,A -85,B 0,C 180,E1 -590.875,E2 -590.875} C_VEL
LIN {X 0,Y 601.423,Z 399.257,A -85,B 0,C 180,E1 -592.051,E2 -592.051} C_VEL
LIN {X 0,Y 601.501,Z 408.141,A -85,B 0,C 180,E1 -594.253,E2 -594.253} C_VEL
LIN {X 0,Y 601.555,Z 420.161,A -85,B 0,C 180,E1 -597.265,E2 -597.265} C_VEL
LIN {X 0,Y 601.556,Z 428.33,A -85,B 0,C 180,E1 -599.456,E2 -599.456} C_VEL
LIN {X 0,Y 601.527,Z 438.268,A -85,B 0,C 180,E1 -602.138,E2 -602.138} C_VEL
LIN {X 0,Y 601.49,Z 448.208,A -85,B 0,C 180,E1 -604.756,E2 -604.756} C_VEL
LIN {X 0,Y 601.46,Z 459.694,A -85,B 0,C 180,E1 -607.713,E2 -607.713} C_VEL
LIN {X 0,Y 601.424,Z 470.929,A -85,B 0,C 180,E1 -610.547,E2 -610.547} C_VEL
LIN {X 0,Y 601.419,Z 480.87,A -85,B 0,C 180,E1 -613.014,E2 -613.014} C_VEL
LIN {X 0,Y 601.407,Z 491.66,A -85,B 0,C 180,E1 -615.655,E2 -615.655} C_VEL
LIN {X 0,Y 601.733,Z 495.192,A -85,B 0,C 180,E1 -615.711,E2 -615.711} C_VEL
LIN {X 0,Y 601.698,Z 510.019,A -85,B 0,C 180,E1 -615.992,E2 -615.992} C_VEL
LIN {X 0,Y 601.654,Z 523.599,A -85,B 0,C 180,E1 -616.387,E2 -616.387} C_VEL
LIN {X 0,Y 601.623,Z 537.071,A -85,B 0,C 180,E1 -616.919,E2 -616.919} C_VEL
LIN {X 0,Y 601.563,Z 548.953,A -85,B 0,C 180,E1 -617.518,E2 -617.518} C_VEL
LIN {X 0,Y 601.534,Z 561.312,A -85,B 0,C 180,E1 -618.288,E2 -618.288} C_VEL
LIN {X 0,Y 601.496,Z 572.301,A -85,B 0,C 180,E1 -619.124,E2 -619.124} C_VEL
LIN {X 0,Y 601.435,Z 582.652,A -85,B 0,C 180,E1 -620.075,E2 -620.075} C_VEL
LIN {X 0,Y 601.411,Z 591.84,A -85,B 0,C 180,E1 -621.093,E2 -621.093} C_VEL
LIN {X 0,Y 601.387,Z 600.623,A -85,B 0,C 180,E1 -622.276,E2 -622.276} C_VEL
LIN {X 0,Y 601.373,Z 607.384,A -85,B 0,C 180,E1 -623.395,E2 -623.395} C_VEL
LIN {X 0,Y 601.352,Z 613.38,A -85,B 0,C 180,E1 -624.635,E2 -624.635} C_VEL
LIN {X 0,Y 601.345,Z 618.301,A -85,B 0,C 180,E1 -625.979,E2 -625.979} C_VEL
LIN {X 0,Y 601.324,Z 621.737,A -85,B 0,C 180,E1 -627.32,E2 -627.32} C_VEL
LIN {X 0,Y 601.346,Z 623.78,A -85,B 0,C 180,E1 -628.661,E2 -628.661} C_VEL
LIN {X 0,Y 601.334,Z 624.496,A -85,B 0,C 180,E1 -630,E2 -630} C_VEL
LIN {X 0,Y 601.343,Z 623.88,A -85,B 0,C 180,E1 -631.339,E2 -631.339} C_VEL
LIN {X 0,Y 601.321,Z 621.929,A -85,B 0,C 180,E1 -632.68,E2 -632.68} C_VEL
LIN {X 0,Y 601.346,Z 618.585,A -85,B 0,C 180,E1 -634.021,E2 -634.021} C_VEL
LIN {X 0,Y 601.355,Z 613.761,A -85,B 0,C 180,E1 -635.365,E2 -635.365} C_VEL
LIN {X 0,Y 601.368,Z 607.89,A -85,B 0,C 180,E1 -636.601,E2 -636.601} C_VEL
LIN {X 0,Y 601.386,Z 601.22,A -85,B 0,C 180,E1 -637.724,E2 -637.724} C_VEL
LIN {X 0,Y 601.411,Z 592.563,A -85,B 0,C 180,E1 -638.907,E2 -638.907} C_VEL
LIN {X 0,Y 601.431,Z 583.515,A -85,B 0,C 180,E1 -639.925,E2 -639.925} C_VEL
LIN {X 0,Y 601.497,Z 573.352,A -85,B 0,C 180,E1 -640.876,E2 -640.876} C_VEL
LIN {X 0,Y 601.549,Z 561.379,A -85,B 0,C 180,E1 -641.798,E2 -641.798} C_VEL
LIN {X 0,Y 601.578,Z 549.031,A -85,B 0,C 180,E1 -642.567,E2 -642.567} C_VEL
LIN {X 0,Y 601.624,Z 537.166,A -85,B 0,C 180,E1 -643.167,E2 -643.167} C_VEL
LIN {X 0,Y 601.663,Z 524.248,A -85,B 0,C 180,E1 -643.681,E2 -643.681} C_VEL
LIN {X 0,Y 601.719,Z 509.943,A -85,B 0,C 180,E1 -644.099,E2 -644.099} C_VEL
LIN {X 0,Y 601.723,Z 495.647,A -85,B 0,C 180,E1 -644.373,E2 -644.373} C_VEL
LIN {X 0,Y 601.369,Z 491.644,A -85,B 0,C 180,E1 -644.44,E2 -644.44} C_VEL
LIN {X 0,Y 601.439,Z 479.815,A -85,B 0,C 180,E1 -647.336,E2 -647.336} C_VEL
LIN {X 0,Y 601.427,Z 468.447,A -85,B 0,C 180,E1 -650.165,E2 -650.165} C_VEL
LIN {X 0,Y 601.456,Z 457.08,A -85,B 0,C 180,E1 -653.045,E2 -653.045} C_VEL
LIN {X 0,Y 601.522,Z 446.081,A -85,B 0,C 180,E1 -655.888,E2 -655.888} C_VEL
LIN {X 0,Y 601.518,Z 435.764,A -85,B 0,C 180,E1 -658.622,E2 -658.622} C_VEL
LIN {X 0,Y 601.571,Z 425.26,A -85,B 0,C 180,E1 -661.478,E2 -661.478} C_VEL
LIN {X 0,Y 601.506,Z 417.025,A -85,B 0,C 180,E1 -663.625,E2 -663.625} C_VEL
LIN {X 0,Y 601.522,Z 405.178,A -85,B 0,C 180,E1 -666.575,E2 -666.575} C_VEL
LIN {X 0,Y 601.418,Z 399.197,A -85,B 0,C 180,E1 -668.055,E2 -668.055} C_VEL
LIN {X 0,Y 601.418,Z 399.198,A -85,B 0,C 180,E1 -670.874,E2 -670.874} C_VEL
LIN {X 0,Y 601.431,Z 399.196,A -85,B 0,C 180,E1 -673.586,E2 -673.586} C_VEL
LIN {X 0,Y 601.453,Z 399.191,A -85,B 0,C 180,E1 -676.425,E2 -676.425} C_VEL
LIN {X 0,Y 601.419,Z 399.199,A -85,B 0,C 180,E1 -679.426,E2 -679.426} C_VEL
LIN {X 0,Y 601.421,Z 399.198,A -85,B 0,C 180,E1 -681.732,E2 -681.732} C_VEL
LIN {X 0,Y 601.409,Z 399.201,A -85,B 0,C 180,E1 -684.247,E2 -684.247} C_VEL
LIN {X 0,Y 601.421,Z 399.199,A -85,B 0,C 180,E1 -686.686,E2 -686.686} C_VEL
LIN {X 0,Y 601.427,Z 399.198,A -85,B 0,C 180,E1 -689.058,E2 -689.058} C_VEL
LIN {X 0,Y 601.436,Z 399.196,A -85,B 0,C 180,E1 -691.373,E2 -691.373} C_VEL
LIN {X 0,Y 601.403,Z 399.199,A -85,B 0,C 180,E1 -693.636,E2 -693.636} C_VEL
LIN {X 0,Y 601.423,Z 399.196,A -85,B 0,C 180,E1 -696.59,E2 -696.59} C_VEL
LIN {X 0,Y 601.433,Z 399.194,A -85,B 0,C 180,E1 -699.478,E2 -699.478} C_VEL
LIN {X 0,Y 601.4,Z 399.201,A -85,B 0,C 180,E1 -702.312,E2 -702.312} C_VEL
LIN {X 0,Y 601.449,Z 399.195,A -85,B 0,C 180,E1 -703.624,E2 -703.624} C_VEL
LIN {X 0,Y 601.815,Z 402.228,A -85,B 0,C 180,E1 -703.709,E2 -703.709} C_VEL
LIN {X 0,Y 601.792,Z 417.47,A -85,B 0,C 180,E1 -704.158,E2 -704.158} C_VEL
LIN {X 0,Y 601.73,Z 430.755,A -85,B 0,C 180,E1 -704.677,E2 -704.677} C_VEL
LIN {X 0,Y 601.66,Z 444.858,A -85,B 0,C 180,E1 -705.368,E2 -705.368} C_VEL
LIN {X 0,Y 601.621,Z 458.77,A -85,B 0,C 180,E1 -706.215,E2 -706.215} C_VEL
LIN {X 0,Y 601.531,Z 471.72,A -85,B 0,C 180,E1 -707.174,E2 -707.174} C_VEL
LIN {X 0,Y 601.488,Z 483.285,A -85,B 0,C 180,E1 -708.201,E2 -708.201} C_VEL
LIN {X 0,Y 601.439,Z 494.488,A -85,B 0,C 180,E1 -709.395,E2 -709.395} C_VEL
LIN {X 0,Y 601.394,Z 503.758,A -85,B 0,C 180,E1 -710.584,E2 -710.584} C_VEL
LIN {X 0,Y 601.399,Z 511.474,A -85,B 0,C 180,E1 -711.77,E2 -711.77} C_VEL
LIN {X 0,Y 601.368,Z 517.875,A -85,B 0,C 180,E1 -712.951,E2 -712.951} C_VEL
LIN {X 0,Y 601.369,Z 523.754,A -85,B 0,C 180,E1 -714.299,E2 -714.299} C_VEL
LIN {X 0,Y 601.332,Z 527.244,A -85,B 0,C 180,E1 -715.307,E2 -715.307} C_VEL
LIN {X 0,Y 601.339,Z 530.786,A -85,B 0,C 180,E1 -716.65,E2 -716.65} C_VEL
LIN {X 0,Y 601.337,Z 533.141,A -85,B 0,C 180,E1 -717.991,E2 -717.991} C_VEL
LIN {X 0,Y 601.332,Z 534.336,A -85,B 0,C 180,E1 -719.33,E2 -719.33} C_VEL
LIN {X 0,Y 601.337,Z 534.362,A -85,B 0,C 180,E1 -720.67,E2 -720.67} C_VEL
LIN {X 0,Y 601.34,Z 533.247,A -85,B 0,C 180,E1 -722.009,E2 -722.009} C_VEL
LIN {X 0,Y 601.341,Z 530.982,A -85,B 0,C 180,E1 -723.35,E2 -723.35} C_VEL
LIN {X 0,Y 601.328,Z 527.525,A -85,B 0,C 180,E1 -724.693,E2 -724.693} C_VEL
LIN {X 0,Y 601.353,Z 522.802,A -85,B 0,C 180,E1 -726.038,E2 -726.038} C_VEL
LIN {X 0,Y 601.366,Z 516.667,A -85,B 0,C 180,E1 -727.386,E2 -727.386} C_VEL
LIN {X 0,Y 601.389,Z 508.942,A -85,B 0,C 180,E1 -728.738,E2 -728.738} C_VEL
LIN {X 0,Y 601.427,Z 500.697,A -85,B 0,C 180,E1 -729.925,E2 -729.925} C_VEL
LIN {X 0,Y 601.461,Z 490.363,A -85,B 0,C 180,E1 -731.164,E2 -731.164} C_VEL
LIN {X 0,Y 601.501,Z 478.779,A -85,B 0,C 180,E1 -732.312,E2 -732.312} C_VEL
LIN {X 0,Y 601.557,Z 467.468,A -85,B 0,C 180,E1 -733.255,E2 -733.255} C_VEL
LIN {X 0,Y 601.624,Z 454.316,A -85,B 0,C 180,E1 -734.167,E2 -734.167} C_VEL
LIN {X 0,Y 601.676,Z 441.743,A -85,B 0,C 180,E1 -734.891,E2 -734.891} C_VEL
LIN {X 0,Y 601.73,Z 427.866,A -85,B 0,C 180,E1 -735.539,E2 -735.539} C_VEL
LIN {X 0,Y 601.812,Z 412.324,A -85,B 0,C 180,E1 -736.102,E2 -736.102} C_VEL
LIN {X 0,Y 601.725,Z 400.489,A -85,B 0,C 180,E1 -736.425,E2 -736.425} C_VEL
LIN {X 0,Y 601.449,Z 399.19,A -85,B 0,C 180,E1 -736.49,E2 -736.49} C_VEL
LIN {X 0,Y 601.42,Z 399.189,A -85,B 0,C 180,E1 -739.099,E2 -739.099} C_VEL
LIN {X 0,Y 601.422,Z 399.198,A -85,B 0,C 180,E1 -741.959,E2 -741.959} C_VEL
LIN {X 0,Y 601.438,Z 399.192,A -85,B 0,C 180,E1 -744.293,E2 -744.293} C_VEL
LIN {X 0,Y 601.449,Z 399.186,A -85,B 0,C 180,E1 -747.111,E2 -747.111} C_VEL
LIN {X 0,Y 601.426,Z 399.191,A -85,B 0,C 180,E1 -749.393,E2 -749.393} C_VEL
LIN {X 0,Y 601.419,Z 399.198,A -85,B 0,C 180,E1 -751.726,E2 -751.726} C_VEL
LIN {X 0,Y 601.429,Z 399.192,A -85,B 0,C 180,E1 -754.118,E2 -754.118} C_VEL
LIN {X 0,Y 601.401,Z 399.191,A -85,B 0,C 180,E1 -756.583,E2 -756.583} C_VEL
LIN {X 0,Y 601.411,Z 399.193,A -85,B 0,C 180,E1 -759.127,E2 -759.127} C_VEL
LIN {X 0,Y 601.427,Z 399.195,A -85,B 0,C 180,E1 -761.765,E2 -761.765} C_VEL
LIN {X 0,Y 601.426,Z 399.188,A -85,B 0,C 180,E1 -764.535,E2 -764.535} C_VEL
LIN {X 0,Y 601.411,Z 399.226,A -85,B 0,C 180,E1 -765.074,E2 -765.074} C_VEL
LIN {X 0,Y 601.371,Z 411.304,A -85,B 0,C 180,E1 -767.823,E2 -767.823} C_VEL
LIN {X 0,Y 601.583,Z 417.976,A -85,B 0,C 180,E1 -769.408,E2 -769.408} C_VEL
LIN {X 0,Y 601.589,Z 424.788,A -85,B 0,C 180,E1 -771.745,E2 -771.745} C_VEL
LIN {X 0,Y 601.571,Z 432.131,A -85,B 0,C 180,E1 -774.258,E2 -774.258} C_VEL
LIN {X 0,Y 601.526,Z 439.474,A -85,B 0,C 180,E1 -776.693,E2 -776.693} C_VEL
LIN {X 0,Y 601.509,Z 448.04,A -85,B 0,C 180,E1 -779.453,E2 -779.453} C_VEL
LIN {X 0,Y 601.503,Z 456.606,A -85,B 0,C 180,E1 -782.137,E2 -782.137} C_VEL
LIN {X 0,Y 601.458,Z 466.396,A -85,B 0,C 180,E1 -785.124,E2 -785.124} C_VEL
LIN {X 0,Y 601.434,Z 476.186,A -85,B 0,C 180,E1 -788.042,E2 -788.042} C_VEL
LIN {X 0,Y 601.413,Z 485.976,A -85,B 0,C 180,E1 -790.901,E2 -790.901} C_VEL
LIN {X 0,Y 601.365,Z 495.766,A -85,B 0,C 180,E1 -793.711,E2 -793.711} C_VEL
LIN {X 0,Y 601.369,Z 502.49,A -85,B 0,C 180,E1 -795.619,E2 -795.619} C_VEL
LIN {X 0,Y 601.739,Z 506.821,A -85,B 0,C 180,E1 -795.69,E2 -795.69} C_VEL
LIN {X 0,Y 601.707,Z 521.033,A -85,B 0,C 180,E1 -795.972,E2 -795.972} C_VEL
LIN {X 0,Y 601.67,Z 533.926,A -85,B 0,C 180,E1 -796.353,E2 -796.353} C_VEL
LIN {X 0,Y 601.626,Z 546.13,A -85,B 0,C 180,E1 -796.833,E2 -796.833} C_VEL
LIN {X 0,Y 601.564,Z 559.777,A -85,B 0,C 180,E1 -797.518,E2 -797.518} C_VEL
LIN {X 0,Y 601.534,Z 571.966,A -85,B 0,C 180,E1 -798.288,E2 -798.288} C_VEL
LIN {X 0,Y 601.486,Z 582.76,A -85,B 0,C 180,E1 -799.117,E2 -799.117} C_VEL
LIN {X 0,Y 601.432,Z 593.085,A -85,B 0,C 180,E1 -800.075,E2 -800.075} C_VEL
LIN {X 0,Y 601.411,Z 602.2,A -85,B 0,C 180,E1 -801.093,E2 -801.093} C_VEL
LIN {X 0,Y 601.386,Z 610.92,A -85,B 0,C 180,E1 -802.276,E2 -802.276} C_VEL
LIN {X 0,Y 601.367,Z 617.646,A -85,B 0,C 180,E1 -803.399,E2 -803.399} C_VEL
LIN {X 0,Y 601.355,Z 623.569,A -85,B 0,C 180,E1 -804.635,E2 -804.635} C_VEL
LIN {X 0,Y 601.343,Z 628.442,A -85,B 0,C 180,E1 -805.979,E2 -805.979} C_VEL
LIN {X 0,Y 601.324,Z 631.831,A -85,B 0,C 180,E1 -807.32,E2 -807.32} C_VEL
LIN {X 0,Y 601.342,Z 633.83,A -85,B 0,C 180,E1 -808.661,E2 -808.661} C_VEL
LIN {X 0,Y 601.333,Z 634.5,A -85,B 0,C 180,E1 -810,E2 -810} C_VEL
LIN {X 0,Y 601.342,Z 633.831,A -85,B 0,C 180,E1 -811.339,E2 -811.339} C_VEL
LIN {X 0,Y 601.324,Z 631.832,A -85,B 0,C 180,E1 -812.68,E2 -812.68} C_VEL
LIN {X 0,Y 601.343,Z 628.443,A -85,B 0,C 180,E1 -814.021,E2 -814.021} C_VEL
LIN {X 0,Y 601.355,Z 623.569,A -85,B 0,C 180,E1 -815.365,E2 -815.365} C_VEL
LIN {X 0,Y 601.372,Z 617.624,A -85,B 0,C 180,E1 -816.605,E2 -816.605} C_VEL
LIN {X 0,Y 601.386,Z 610.92,A -85,B 0,C 180,E1 -817.724,E2 -817.724} C_VEL
LIN {X 0,Y 601.411,Z 602.198,A -85,B 0,C 180,E1 -818.907,E2 -818.907} C_VEL
LIN {X 0,Y 601.432,Z 593.082,A -85,B 0,C 180,E1 -819.925,E2 -819.925} C_VEL
LIN {X 0,Y 601.497,Z 582.831,A -85,B 0,C 180,E1 -820.876,E2 -820.876} C_VEL
LIN {X 0,Y 601.534,Z 571.969,A -85,B 0,C 180,E1 -821.712,E2 -821.712} C_VEL
LIN {X 0,Y 601.564,Z 559.776,A -85,B 0,C 180,E1 -822.482,E2 -822.482} C_VEL
LIN {X 0,Y 601.626,Z 546.13,A -85,B 0,C 180,E1 -823.167,E2 -823.167} C_VEL
LIN {X 0,Y 601.653,Z 532.899,A -85,B 0,C 180,E1 -823.681,E2 -823.681} C_VEL
LIN {X 0,Y 601.717,Z 518.643,A -85,B 0,C 180,E1 -824.084,E2 -824.084} C_VEL
LIN {X 0,Y 601.727,Z 504.43,A -85,B 0,C 180,E1 -824.345,E2 -824.345} C_VEL
LIN {X 0,Y 601.376,Z 502.474,A -85,B 0,C 180,E1 -824.386,E2 -824.386} C_VEL
LIN {X 0,Y 601.383,Z 493.319,A -85,B 0,C 180,E1 -826.987,E2 -826.987} C_VEL
LIN {X 0,Y 601.413,Z 483.529,A -85,B 0,C 180,E1 -829.809,E2 -829.809} C_VEL
LIN {X 0,Y 601.418,Z 473.739,A -85,B 0,C 180,E1 -832.683,E2 -832.683} C_VEL
LIN {X 0,Y 601.449,Z 465.172,A -85,B 0,C 180,E1 -835.246,E2 -835.246} C_VEL
LIN {X 0,Y 601.503,Z 456.606,A -85,B 0,C 180,E1 -837.863,E2 -837.863} C_VEL
LIN {X 0,Y 601.538,Z 446.816,A -85,B 0,C 180,E1 -840.935,E2 -840.935} C_VEL
LIN {X 0,Y 601.566,Z 437.496,A -85,B 0,C 180,E1 -843.954,E2 -843.954} C_VEL
LIN {X 0,Y 601.578,Z 429.683,A -85,B 0,C 180,E1 -846.571,E2 -846.571} C_VEL
LIN {X 0,Y 601.605,Z 422.341,A -85,B 0,C 180,E1 -849.112,E2 -849.112} C_VEL
LIN {X 0,Y 601.577,Z 414.961,A -85,B 0,C 180,E1 -851.609,E2 -851.609} C_VEL
LIN {X 0,Y 601.613,Z 406.341,A -85,B 0,C 180,E1 -854.553,E2 -854.553} C_VEL
LIN {X 0,Y 601.548,Z 399.842,A -85,B 0,C 180,E1 -856.885,E2 -856.885} C_VEL
LIN {X 0,Y 601.404,Z 399.199,A -85,B 0,C 180,E1 -857.215,E2 -857.215} C_VEL
LIN {X 0,Y 601.403,Z 399.196,A -85,B 0,C 180,E1 -860.004,E2 -860.004} C_VEL
LIN {X 0,Y 601.437,Z 399.194,A -85,B 0,C 180,E1 -862.618,E2 -862.618} C_VEL
LIN {X 0,Y 601.415,Z 399.196,A -85,B 0,C 180,E1 -865.068,E2 -865.068} C_VEL
LIN {X 0,Y 601.434,Z 399.192,A -85,B 0,C 180,E1 -867.484,E2 -867.484} C_VEL
LIN {X 0,Y 601.431,Z 399.197,A -85,B 0,C 180,E1 -869.851,E2 -869.851} C_VEL
LIN {X 0,Y 601.421,Z 399.195,A -85,B 0,C 180,E1 -872.637,E2 -872.637} C_VEL
LIN {X 0,Y 601.404,Z 399.195,A -85,B 0,C 180,E1 -875.122,E2 -875.122} C_VEL
LIN {X 0,Y 601.418,Z 399.199,A -85,B 0,C 180,E1 -877.394,E2 -877.394} C_VEL
LIN {X 0,Y 601.407,Z 399.197,A -85,B 0,C 180,E1 -880.191,E2 -880.191} C_VEL
LIN {X 0,Y 601.437,Z 399.192,A -85,B 0,C 180,E1 -883.014,E2 -883.014} C_VEL
LIN {X 0,Y 601.423,Z 399.193,A -85,B 0,C 180,E1 -885.908,E2 -885.908} C_VEL
LIN {X 0,Y 601.437,Z 399.191,A -85,B 0,C 180,E1 -888.542,E2 -888.542} C_VEL
LIN {X 0,Y 601.418,Z 399.195,A -85,B 0,C 180,E1 -891.262,E2 -891.262} C_VEL
LIN {X 0,Y 601.42,Z 399.199,A -85,B 0,C 180,E1 -893.963,E2 -893.963} C_VEL
LIN {X 0,Y 601.437,Z 399.192,A -85,B 0,C 180,E1 -896.651,E2 -896.651} C_VEL
LIN {X 0,Y 601.449,Z 399.189,A -85,B 0,C 180,E1 -899.331,E2 -899.331} C_VEL
LIN {X 0,Y 601.419,Z 399.193,A -85,B 0,C 180,E1 -902.009,E2 -902.009} C_VEL
LIN {X 0,Y 601.427,Z 399.196,A -85,B 0,C 180,E1 -904.692,E2 -904.692} C_VEL
LIN {X 0,Y 601.441,Z 399.195,A -85,B 0,C 180,E1 -907.385,E2 -907.385} C_VEL
LIN {X 0,Y 601.43,Z 399.193,A -85,B 0,C 180,E1 -910.095,E2 -910.095} C_VEL
LIN {X 0,Y 601.411,Z 399.196,A -85,B 0,C 180,E1 -912.376,E2 -912.376} C_VEL
LIN {X 0,Y 600.745,Z 399.278,A -85,B 0,C 180,E1 -912.935,E2 -912.935} C_VEL
LIN {X 0,Y 597.897,Z 399.635,A -85,B 0,C 180,E1 -913.843,E2 -913.843} C_VEL
LIN {X 0,Y 595.489,Z 399.938,A -85,B 0,C 180,E1 -914.573,E2 -914.573} C_VEL
LIN {X 0,Y 594.451,Z 400.066,A -85,B 0,C 180,E1 -915.137,E2 -915.137} C_VEL
LIN {X 0,Y 594.364,Z 400.074,A -85,B 0,C 180,E1 -915.328,E2 -915.328} C_VEL
LIN {X 0,Y 594.392,Z 400.069,A -85,B 0,C 180,E1 -917.193,E2 -917.193} C_VEL
LIN {X 0,Y 594.378,Z 400.071,A -85,B 0,C 180,E1 -920.054,E2 -920.054} C_VEL
LIN {X 0,Y 594.36,Z 400.073,A -85,B 0,C 180,E1 -922.968,E2 -922.968} C_VEL
LIN {X 0,Y 594.379,Z 400.072,A -85,B 0,C 180,E1 -925.193,E2 -925.193} C_VEL
LIN {X 0,Y 594.389,Z 400.07,A -85,B 0,C 180,E1 -927.527,E2 -927.527} C_VEL
LIN {X 0,Y 594.389,Z 400.072,A -85,B 0,C 180,E1 -930.328,E2 -930.328} C_VEL
LIN {X 0,Y 594.381,Z 400.074,A -85,B 0,C 180,E1 -932.95,E2 -932.95} C_VEL
LIN {X 0,Y 594.35,Z 400.074,A -85,B 0,C 180,E1 -935.409,E2 -935.409} C_VEL
LIN {X 0,Y 594.39,Z 400.071,A -85,B 0,C 180,E1 -937.941,E2 -937.941} C_VEL
LIN {X 0,Y 594.379,Z 400.074,A -85,B 0,C 180,E1 -940.822,E2 -940.822} C_VEL
LIN {X 0,Y 594.386,Z 400.073,A -85,B 0,C 180,E1 -943.841,E2 -943.841} C_VEL
LIN {X 0,Y 594.368,Z 400.078,A -85,B 0,C 180,E1 -946.701,E2 -946.701} C_VEL
LIN {X 0,Y 594.372,Z 400.075,A -85,B 0,C 180,E1 -949.433,E2 -949.433} C_VEL
LIN {X 0,Y 594.417,Z 400.245,A -85,B 0,C 180,E1 -951.954,E2 -951.954} C_VEL
LIN {X 0,Y 594.527,Z 407.49,A -85,B 0,C 180,E1 -953.768,E2 -953.768} C_VEL
LIN {X 0,Y 594.518,Z 418.884,A -85,B 0,C 180,E1 -956.654,E2 -956.654} C_VEL
LIN {X 0,Y 594.6,Z 429.751,A -85,B 0,C 180,E1 -959.453,E2 -959.453} C_VEL
LIN {X 0,Y 594.552,Z 440.721,A -85,B 0,C 180,E1 -962.443,E2 -962.443} C_VEL
LIN {X 0,Y 594.483,Z 451.052,A -85,B 0,C 180,E1 -965.186,E2 -965.186} C_VEL
LIN {X 0,Y 594.422,Z 462.411,A -85,B 0,C 180,E1 -968.134,E2 -968.134} C_VEL
LIN {X 0,Y 594.387,Z 473.953,A -85,B 0,C 180,E1 -971.07,E2 -971.07} C_VEL
LIN {X 0,Y 594.322,Z 483.713,A -85,B 0,C 180,E1 -973.512,E2 -973.512} C_VEL
LIN {X 0,Y 594.349,Z 491.677,A -85,B 0,C 180,E1 -975.481,E2 -975.481} C_VEL
LIN {X 0,Y 594.863,Z 496.332,A -85,B 0,C 180,E1 -975.558,E2 -975.558} C_VEL
LIN {X 0,Y 594.817,Z 511.184,A -85,B 0,C 180,E1 -975.854,E2 -975.854} C_VEL
LIN {X 0,Y 594.749,Z 524.761,A -85,B 0,C 180,E1 -976.264,E2 -976.264} C_VEL
LIN {X 0,Y 594.683,Z 538.983,A -85,B 0,C 180,E1 -976.85,E2 -976.85} C_VEL
LIN {X 0,Y 594.592,Z 551.954,A -85,B 0,C 180,E1 -977.543,E2 -977.543} C_VEL
LIN {X 0,Y 594.507,Z 563.714,A -85,B 0,C 180,E1 -978.32,E2 -978.32} C_VEL
LIN {X 0,Y 594.474,Z 575.43,A -85,B 0,C 180,E1 -979.269,E2 -979.269} C_VEL
LIN {X 0,Y 594.392,Z 585.912,A -85,B 0,C 180,E1 -980.3,E2 -980.3} C_VEL
LIN {X 0,Y 594.355,Z 594.566,A -85,B 0,C 180,E1 -981.329,E2 -981.329} C_VEL
LIN {X 0,Y 594.314,Z 602.846,A -85,B 0,C 180,E1 -982.526,E2 -982.526} C_VEL
LIN {X 0,Y 594.271,Z 609.005,A -85,B 0,C 180,E1 -983.62,E2 -983.62} C_VEL
LIN {X 0,Y 594.246,Z 614.789,A -85,B 0,C 180,E1 -984.911,E2 -984.911} C_VEL
LIN {X 0,Y 594.261,Z 618.304,A -85,B 0,C 180,E1 -985.931,E2 -985.931} C_VEL
LIN {X 0,Y 594.224,Z 621.74,A -85,B 0,C 180,E1 -987.288,E2 -987.288} C_VEL
LIN {X 0,Y 594.245,Z 623.783,A -85,B 0,C 180,E1 -988.645,E2 -988.645} C_VEL
LIN {X 0,Y 594.235,Z 624.496,A -85,B 0,C 180,E1 -990,E2 -990} C_VEL
LIN {X 0,Y 594.242,Z 623.878,A -85,B 0,C 180,E1 -991.355,E2 -991.355} C_VEL
LIN {X 0,Y 594.222,Z 621.93,A -85,B 0,C 180,E1 -992.712,E2 -992.712} C_VEL
LIN {X 0,Y 594.262,Z 618.584,A -85,B 0,C 180,E1 -994.069,E2 -994.069} C_VEL
LIN {X 0,Y 594.275,Z 613.761,A -85,B 0,C 180,E1 -995.429,E2 -995.429} C_VEL
LIN {X 0,Y 594.277,Z 608.383,A -85,B 0,C 180,E1 -996.587,E2 -996.587} C_VEL
LIN {X 0,Y 594.316,Z 601.218,A -85,B 0,C 180,E1 -997.816,E2 -997.816} C_VEL
LIN {X 0,Y 594.368,Z 592.561,A -85,B 0,C 180,E1 -999.014,E2 -999.014} C_VEL
LIN {X 0,Y 594.399,Z 583.511,A -85,B 0,C 180,E1 -1000.044,E2 -1000.044} C_VEL
LIN {X 0,Y 594.478,Z 573.227,A -85,B 0,C 180,E1 -1001.017,E2 -1001.017} C_VEL
LIN {X 0,Y 594.572,Z 561.374,A -85,B 0,C 180,E1 -1001.938,E2 -1001.938} C_VEL
LIN {X 0,Y 594.605,Z 549.023,A -85,B 0,C 180,E1 -1002.717,E2 -1002.717} C_VEL
LIN {X 0,Y 594.683,Z 537.16,A -85,B 0,C 180,E1 -1003.324,E2 -1003.324} C_VEL
LIN {X 0,Y 594.757,Z 523.53,A -85,B 0,C 180,E1 -1003.867,E2 -1003.867} C_VEL
LIN {X 0,Y 594.829,Z 509.427,A -85,B 0,C 180,E1 -1004.278,E2 -1004.278} C_VEL
LIN {X 0,Y 594.852,Z 494.863,A -85,B 0,C 180,E1 -1004.554,E2 -1004.554} C_VEL
LIN {X 0,Y 594.317,Z 491.615,A -85,B 0,C 180,E1 -1004.621,E2 -1004.621} C_VEL
LIN {X 0,Y 594.403,Z 479.812,A -85,B 0,C 180,E1 -1007.548,E2 -1007.548} C_VEL
LIN {X 0,Y 594.387,Z 468.445,A -85,B 0,C 180,E1 -1010.414,E2 -1010.414} C_VEL
LIN {X 0,Y 594.436,Z 458.498,A -85,B 0,C 180,E1 -1012.964,E2 -1012.964} C_VEL
LIN {X 0,Y 594.543,Z 447.13,A -85,B 0,C 180,E1 -1015.936,E2 -1015.936} C_VEL
LIN {X 0,Y 594.547,Z 437.182,A -85,B 0,C 180,E1 -1018.603,E2 -1018.603} C_VEL
LIN {X 0,Y 594.603,Z 427.147,A -85,B 0,C 180,E1 -1021.337,E2 -1021.337} C_VEL
LIN {X 0,Y 594.474,Z 416.072,A -85,B 0,C 180,E1 -1024.151,E2 -1024.151} C_VEL
LIN {X 0,Y 594.551,Z 404.487,A -85,B 0,C 180,E1 -1027.075,E2 -1027.075} C_VEL
LIN {X 0,Y 594.405,Z 400.072,A -85,B 0,C 180,E1 -1028.208,E2 -1028.208} C_VEL
LIN {X 0,Y 594.38,Z 400.075,A -85,B 0,C 180,E1 -1030.822,E2 -1030.822} C_VEL
LIN {X 0,Y 594.369,Z 400.076,A -85,B 0,C 180,E1 -1033.299,E2 -1033.299} C_VEL
LIN {X 0,Y 594.386,Z 400.073,A -85,B 0,C 180,E1 -1036.159,E2 -1036.159} C_VEL
LIN {X 0,Y 594.381,Z 400.074,A -85,B 0,C 180,E1 -1039.178,E2 -1039.178} C_VEL
LIN {X 0,Y 594.388,Z 400.073,A -85,B 0,C 180,E1 -1042.059,E2 -1042.059} C_VEL
LIN {X 0,Y 594.356,Z 400.076,A -85,B 0,C 180,E1 -1044.676,E2 -1044.676} C_VEL
LIN {X 0,Y 594.381,Z 400.073,A -85,B 0,C 180,E1 -1047.088,E2 -1047.088} C_VEL
LIN {X 0,Y 594.403,Z 400.068,A -85,B 0,C 180,E1 -1049.669,E2 -1049.669} C_VEL
LIN {X 0,Y 594.377,Z 400.075,A -85,B 0,C 180,E1 -1052.539,E2 -1052.539} C_VEL
LIN {X 0,Y 594.378,Z 400.074,A -85,B 0,C 180,E1 -1054.807,E2 -1054.807} C_VEL
LIN {X 0,Y 594.368,Z 400.075,A -85,B 0,C 180,E1 -1057.265,E2 -1057.265} C_VEL
LIN {X 0,Y 594.377,Z 400.076,A -85,B 0,C 180,E1 -1059.946,E2 -1059.946} C_VEL
LIN {X 0,Y 594.392,Z 400.07,A -85,B 0,C 180,E1 -1062.807,E2 -1062.807} C_VEL
LIN {X 0,Y 594.408,Z 400.071,A -85,B 0,C 180,E1 -1063.446,E2 -1063.446} C_VEL
LIN {X 0,Y 594.99,Z 402.864,A -85,B 0,C 180,E1 -1063.531,E2 -1063.531} C_VEL
LIN {X 0,Y 594.954,Z 417.497,A -85,B 0,C 180,E1 -1063.971,E2 -1063.971} C_VEL
LIN {X 0,Y 594.847,Z 430.764,A -85,B 0,C 180,E1 -1064.496,E2 -1064.496} C_VEL
LIN {X 0,Y 594.774,Z 444.875,A -85,B 0,C 180,E1 -1065.195,E2 -1065.195} C_VEL
LIN {X 0,Y 594.682,Z 459.133,A -85,B 0,C 180,E1 -1066.075,E2 -1066.075} C_VEL
LIN {X 0,Y 594.56,Z 471.724,A -85,B 0,C 180,E1 -1067.021,E2 -1067.021} C_VEL
LIN {X 0,Y 594.466,Z 483.294,A -85,B 0,C 180,E1 -1068.06,E2 -1068.06} C_VEL
LIN {X 0,Y 594.401,Z 494.496,A -85,B 0,C 180,E1 -1069.267,E2 -1069.267} C_VEL
LIN {X 0,Y 594.341,Z 503.759,A -85,B 0,C 180,E1 -1070.471,E2 -1070.471} C_VEL
LIN {X 0,Y 594.322,Z 511.479,A -85,B 0,C 180,E1 -1071.671,E2 -1071.671} C_VEL
LIN {X 0,Y 594.293,Z 517.881,A -85,B 0,C 180,E1 -1072.867,E2 -1072.867} C_VEL
LIN {X 0,Y 594.295,Z 523.754,A -85,B 0,C 180,E1 -1074.231,E2 -1074.231} C_VEL
LIN {X 0,Y 594.234,Z 527.248,A -85,B 0,C 180,E1 -1075.251,E2 -1075.251} C_VEL
LIN {X 0,Y 594.258,Z 530.784,A -85,B 0,C 180,E1 -1076.61,E2 -1076.61} C_VEL
LIN {X 0,Y 594.236,Z 533.143,A -85,B 0,C 180,E1 -1077.967,E2 -1077.967} C_VEL
LIN {X 0,Y 594.233,Z 534.334,A -85,B 0,C 180,E1 -1079.322,E2 -1079.322} C_VEL
LIN {X 0,Y 594.237,Z 534.363,A -85,B 0,C 180,E1 -1080.678,E2 -1080.678} C_VEL
LIN {X 0,Y 594.239,Z 533.249,A -85,B 0,C 180,E1 -1082.033,E2 -1082.033} C_VEL
LIN {X 0,Y 594.26,Z 530.98,A -85,B 0,C 180,E1 -1083.39,E2 -1083.39} C_VEL
LIN {X 0,Y 594.231,Z 527.524,A -85,B 0,C 180,E1 -1084.749,E2 -1084.749} C_VEL
LIN {X 0,Y 594.276,Z 522.803,A -85,B 0,C 180,E1 -1086.11,E2 -1086.11} C_VEL
LIN {X 0,Y 594.288,Z 516.663,A -85,B 0,C 180,E1 -1087.474,E2 -1087.474} C_VEL
LIN {X 0,Y 594.332,Z 508.931,A -85,B 0,C 180,E1 -1088.843,E2 -1088.843} C_VEL
LIN {X 0,Y 594.387,Z 500.686,A -85,B 0,C 180,E1 -1090.044,E2 -1090.044} C_VEL
LIN {X 0,Y 594.432,Z 490.975,A -85,B 0,C 180,E1 -1091.229,E2 -1091.229} C_VEL
LIN {X 0,Y 594.513,Z 480.666,A -85,B 0,C 180,E1 -1092.286,E2 -1092.286} C_VEL
LIN {X 0,Y 594.576,Z 468.561,A -85,B 0,C 180,E1 -1093.326,E2 -1093.326} C_VEL
LIN {X 0,Y 594.674,Z 456.726,A -85,B 0,C 180,E1 -1094.178,E2 -1094.178} C_VEL
LIN {X 0,Y 594.773,Z 443.353,A -85,B 0,C 180,E1 -1094.98,E2 -1094.98} C_VEL
LIN {X 0,Y 594.861,Z 428.863,A -85,B 0,C 180,E1 -1095.68,E2 -1095.68} C_VEL
LIN {X 0,Y 594.958,Z 413.675,A -85,B 0,C 180,E1 -1096.249,E2 -1096.249} C_VEL
LIN {X 0,Y 594.928,Z 401.99,A -85,B 0,C 180,E1 -1096.582,E2 -1096.582} C_VEL
LIN {X 0,Y 594.404,Z 400.067,A -85,B 0,C 180,E1 -1096.656,E2 -1096.656} C_VEL
LIN {X 0,Y 594.371,Z 400.068,A -85,B 0,C 180,E1 -1099.334,E2 -1099.334} C_VEL
LIN {X 0,Y 594.371,Z 400.07,A -85,B 0,C 180,E1 -1101.503,E2 -1101.503} C_VEL
LIN {X 0,Y 594.391,Z 400.068,A -85,B 0,C 180,E1 -1104.446,E2 -1104.446} C_VEL
LIN {X 0,Y 594.386,Z 400.066,A -85,B 0,C 180,E1 -1106.699,E2 -1106.699} C_VEL
LIN {X 0,Y 594.384,Z 400.066,A -85,B 0,C 180,E1 -1108.998,E2 -1108.998} C_VEL
LIN {X 0,Y 594.396,Z 400.072,A -85,B 0,C 180,E1 -1111.645,E2 -1111.645} C_VEL
LIN {X 0,Y 594.38,Z 400.066,A -85,B 0,C 180,E1 -1114.58,E2 -1114.58} C_VEL
LIN {X 0,Y 594.391,Z 400.074,A -85,B 0,C 180,E1 -1117.608,E2 -1117.608} C_VEL
LIN {X 0,Y 594.37,Z 400.067,A -85,B 0,C 180,E1 -1120.567,E2 -1120.567} C_VEL
LIN {X 0,Y 594.382,Z 400.072,A -85,B 0,C 180,E1 -1123.298,E2 -1123.298} C_VEL
LIN {X 0,Y 594.354,Z 400.141,A -85,B 0,C 180,E1 -1125.113,E2 -1125.113} C_VEL
LIN {X 0,Y 594.289,Z 412.211,A -85,B 0,C 180,E1 -1127.913,E2 -1127.913} C_VEL
LIN {X 0,Y 594.63,Z 421.727,A -85,B 0,C 180,E1 -1130.196,E2 -1130.196} C_VEL
LIN {X 0,Y 594.641,Z 429.684,A -85,B 0,C 180,E1 -1132.932,E2 -1132.932} C_VEL
LIN {X 0,Y 594.61,Z 438.201,A -85,B 0,C 180,E1 -1135.829,E2 -1135.829} C_VEL
LIN {X 0,Y 594.511,Z 446.816,A -85,B 0,C 180,E1 -1138.658,E2 -1138.658} C_VEL
LIN {X 0,Y 594.508,Z 455.401,A -85,B 0,C 180,E1 -1141.401,E2 -1141.401} C_VEL
LIN {X 0,Y 594.442,Z 463.949,A -85,B 0,C 180,E1 -1144.059,E2 -1144.059} C_VEL
LIN {X 0,Y 594.42,Z 472.515,A -85,B 0,C 180,E1 -1146.667,E2 -1146.667} C_VEL
LIN {X 0,Y 594.38,Z 482.305,A -85,B 0,C 180,E1 -1149.585,E2 -1149.585} C_VEL
LIN {X 0,Y 594.333,Z 492.095,A -85,B 0,C 180,E1 -1152.45,E2 -1152.45} C_VEL
LIN {X 0,Y 594.304,Z 502.486,A -85,B 0,C 180,E1 -1155.443,E2 -1155.443} C_VEL
LIN {X 0,Y 594.858,Z 507.02,A -85,B 0,C 180,E1 -1155.523,E2 -1155.523} C_VEL
LIN {X 0,Y 594.815,Z 521.926,A -85,B 0,C 180,E1 -1155.827,E2 -1155.827} C_VEL
LIN {X 0,Y 594.751,Z 536.006,A -85,B 0,C 180,E1 -1156.264,E2 -1156.264} C_VEL
LIN {X 0,Y 594.673,Z 549.89,A -85,B 0,C 180,E1 -1156.85,E2 -1156.85} C_VEL
LIN {X 0,Y 594.592,Z 562.687,A -85,B 0,C 180,E1 -1157.543,E2 -1157.543} C_VEL
LIN {X 0,Y 594.514,Z 575.476,A -85,B 0,C 180,E1 -1158.407,E2 -1158.407} C_VEL
LIN {X 0,Y 594.474,Z 585.936,A -85,B 0,C 180,E1 -1159.269,E2 -1159.269} C_VEL
LIN {X 0,Y 594.391,Z 596.333,A -85,B 0,C 180,E1 -1160.3,E2 -1160.3} C_VEL
LIN {X 0,Y 594.355,Z 604.91,A -85,B 0,C 180,E1 -1161.329,E2 -1161.329} C_VEL
LIN {X 0,Y 594.314,Z 613.117,A -85,B 0,C 180,E1 -1162.526,E2 -1162.526} C_VEL
LIN {X 0,Y 594.27,Z 619.229,A -85,B 0,C 180,E1 -1163.619,E2 -1163.619} C_VEL
LIN {X 0,Y 594.248,Z 624.964,A -85,B 0,C 180,E1 -1164.911,E2 -1164.911} C_VEL
LIN {X 0,Y 594.259,Z 628.443,A -85,B 0,C 180,E1 -1165.931,E2 -1165.931} C_VEL
LIN {X 0,Y 594.224,Z 631.832,A -85,B 0,C 180,E1 -1167.288,E2 -1167.288} C_VEL
LIN {X 0,Y 594.242,Z 633.83,A -85,B 0,C 180,E1 -1168.645,E2 -1168.645} C_VEL
LIN {X 0,Y 594.234,Z 634.5,A -85,B 0,C 180,E1 -1170,E2 -1170} C_VEL
LIN {X 0,Y 594.242,Z 633.831,A -85,B 0,C 180,E1 -1171.355,E2 -1171.355} C_VEL
LIN {X 0,Y 594.224,Z 631.833,A -85,B 0,C 180,E1 -1172.712,E2 -1172.712} C_VEL
LIN {X 0,Y 594.259,Z 628.444,A -85,B 0,C 180,E1 -1174.069,E2 -1174.069} C_VEL
LIN {X 0,Y 594.275,Z 623.571,A -85,B 0,C 180,E1 -1175.429,E2 -1175.429} C_VEL
LIN {X 0,Y 594.3,Z 618.036,A -85,B 0,C 180,E1 -1176.607,E2 -1176.607} C_VEL
LIN {X 0,Y 594.316,Z 610.921,A -85,B 0,C 180,E1 -1177.816,E2 -1177.816} C_VEL
LIN {X 0,Y 594.369,Z 602.199,A -85,B 0,C 180,E1 -1179.014,E2 -1179.014} C_VEL
LIN {X 0,Y 594.4,Z 593.083,A -85,B 0,C 180,E1 -1180.044,E2 -1180.044} C_VEL
LIN {X 0,Y 594.478,Z 582.702,A -85,B 0,C 180,E1 -1181.018,E2 -1181.018} C_VEL
LIN {X 0,Y 594.575,Z 570.703,A -85,B 0,C 180,E1 -1181.938,E2 -1181.938} C_VEL
LIN {X 0,Y 594.605,Z 558.213,A -85,B 0,C 180,E1 -1182.717,E2 -1182.717} C_VEL
LIN {X 0,Y 594.689,Z 546.134,A -85,B 0,C 180,E1 -1183.324,E2 -1183.324} C_VEL
LIN {X 0,Y 594.779,Z 532.189,A -85,B 0,C 180,E1 -1183.866,E2 -1183.866} C_VEL
LIN {X 0,Y 594.816,Z 518.308,A -85,B 0,C 180,E1 -1184.259,E2 -1184.259} C_VEL
LIN {X 0,Y 594.73,Z 504.784,A -85,B 0,C 180,E1 -1184.512,E2 -1184.512} C_VEL
LIN {X 0,Y 594.339,Z 502.478,A -85,B 0,C 180,E1 -1184.559,E2 -1184.559} C_VEL
LIN {X 0,Y 594.333,Z 492.095,A -85,B 0,C 180,E1 -1187.55,E2 -1187.55} C_VEL
LIN {X 0,Y 594.381,Z 482.305,A -85,B 0,C 180,E1 -1190.415,E2 -1190.415} C_VEL
LIN {X 0,Y 594.42,Z 472.515,A -85,B 0,C 180,E1 -1193.333,E2 -1193.333} C_VEL
LIN {X 0,Y 594.468,Z 462.7,A -85,B 0,C 180,E1 -1196.325,E2 -1196.325} C_VEL
LIN {X 0,Y 594.509,Z 454.159,A -85,B 0,C 180,E1 -1198.992,E2 -1198.992} C_VEL
LIN {X 0,Y 594.534,Z 445.811,A -85,B 0,C 180,E1 -1201.667,E2 -1201.667} C_VEL
LIN {X 0,Y 594.616,Z 437.026,A -85,B 0,C 180,E1 -1204.564,E2 -1204.564} C_VEL
LIN {X 0,Y 594.641,Z 429.683,A -85,B 0,C 180,E1 -1207.068,E2 -1207.068} C_VEL
LIN {X 0,Y 594.656,Z 421.802,A -85,B 0,C 180,E1 -1209.807,E2 -1209.807} C_VEL
LIN {X 0,Y 594.605,Z 414.169,A -85,B 0,C 180,E1 -1212.355,E2 -1212.355} C_VEL
LIN {X 0,Y 594.684,Z 406.13,A -85,B 0,C 180,E1 -1215.16,E2 -1215.16} C_VEL
LIN {X 0,Y 594.653,Z 401.83,A -85,B 0,C 180,E1 -1216.726,E2 -1216.726} C_VEL
LIN {X 0,Y 594.393,Z 400.072,A -85,B 0,C 180,E1 -1217.438,E2 -1217.438} C_VEL
LIN {X 0,Y 594.374,Z 400.072,A -85,B 0,C 180,E1 -1220.319,E2 -1220.319} C_VEL
LIN {X 0,Y 594.386,Z 400.07,A -85,B 0,C 180,E1 -1222.913,E2 -1222.913} C_VEL
LIN {X 0,Y 594.385,Z 400.07,A -85,B 0,C 180,E1 -1225.861,E2 -1225.861} C_VEL
LIN {X 0,Y 594.373,Z 400.074,A -85,B 0,C 180,E1 -1228.65,E2 -1228.65} C_VEL
LIN {X 0,Y 594.387,Z 400.071,A -85,B 0,C 180,E1 -1231.042,E2 -1231.042} C_VEL
LIN {X 0,Y 594.389,Z 400.069,A -85,B 0,C 180,E1 -1233.977,E2 -1233.977} C_VEL
LIN {X 0,Y 594.395,Z 400.07,A -85,B 0,C 180,E1 -1236.296,E2 -1236.296} C_VEL
LIN {X 0,Y 594.405,Z 400.068,A -85,B 0,C 180,E1 -1239.224,E2 -1239.224} C_VEL
LIN {X 0,Y 594.383,Z 400.074,A -85,B 0,C 180,E1 -1242.096,E2 -1242.096} C_VEL
LIN {X 0,Y 594.37,Z 400.071,A -85,B 0,C 180,E1 -1244.219,E2 -1244.219} C_VEL
LIN {X 0,Y 594.38,Z 400.073,A -85,B 0,C 180,E1 -1246.321,E2 -1246.321} C_VEL
LIN {X 0,Y 594.378,Z 400.072,A -85,B 0,C 180,E1 -1249.095,E2 -1249.095} C_VEL
LIN {X 0,Y 594.383,Z 400.069,A -85,B 0,C 180,E1 -1251.843,E2 -1251.843} C_VEL
LIN {X 0,Y 594.376,Z 400.075,A -85,B 0,C 180,E1 -1253.891,E2 -1253.891} C_VEL
LIN {X 0,Y 594.387,Z 400.07,A -85,B 0,C 180,E1 -1256.611,E2 -1256.611} C_VEL
LIN {X 0,Y 594.42,Z 400.065,A -85,B 0,C 180,E1 -1259.323,E2 -1259.323} C_VEL
LIN {X 0,Y 594.391,Z 400.068,A -85,B 0,C 180,E1 -1262.033,E2 -1262.033} C_VEL
LIN {X 0,Y 594.396,Z 400.071,A -85,B 0,C 180,E1 -1264.748,E2 -1264.748} C_VEL
LIN {X 0,Y 594.395,Z 400.074,A -85,B 0,C 180,E1 -1267.473,E2 -1267.473} C_VEL
LIN {X 0,Y 594.391,Z 400.07,A -85,B 0,C 180,E1 -1270.216,E2 -1270.216} C_VEL
LIN {X 0,Y 594.366,Z 400.072,A -85,B 0,C 180,E1 -1272.983,E2 -1272.983} C_VEL
LIN {X 0,Y 594.364,Z 400.074,A -85,B 0,C 180,E1 -1275.328,E2 -1275.328} C_VEL
LIN {X 0,Y 593.689,Z 400.157,A -85,B 0,C 180,E1 -1275.894,E2 -1275.894} C_VEL
LIN {X 0,Y 590.822,Z 400.516,A -85,B 0,C 180,E1 -1276.812,E2 -1276.812} C_VEL
LIN {X 0,Y 588.411,Z 400.819,A -85,B 0,C 180,E1 -1277.55,E2 -1277.55} C_VEL
LIN {X 0,Y 587.389,Z 400.945,A -85,B 0,C 180,E1 -1278.12,E2 -1278.12} C_VEL
LIN {X 0,Y 587.312,Z 400.952,A -85,B 0,C 180,E1 -1278.313,E2 -1278.313} C_VEL
LIN {X 0,Y 587.333,Z 400.954,A -85,B 0,C 180,E1 -1281.038,E2 -1281.038} C_VEL
LIN {X 0,Y 587.318,Z 400.949,A -85,B 0,C 180,E1 -1283.259,E2 -1283.259} C_VEL
LIN {X 0,Y 587.339,Z 400.952,A -85,B 0,C 180,E1 -1285.517,E2 -1285.517} C_VEL
LIN {X 0,Y 587.35,Z 400.946,A -85,B 0,C 180,E1 -1287.818,E2 -1287.818} C_VEL
LIN {X 0,Y 587.341,Z 400.948,A -85,B 0,C 180,E1 -1290.51,E2 -1290.51} C_VEL
LIN {X 0,Y 587.336,Z 400.95,A -85,B 0,C 180,E1 -1293.397,E2 -1293.397} C_VEL
LIN {X 0,Y 587.292,Z 400.956,A -85,B 0,C 180,E1 -1295.9,E2 -1295.9} C_VEL
LIN {X 0,Y 587.333,Z 400.948,A -85,B 0,C 180,E1 -1298.479,E2 -1298.479} C_VEL
LIN {X 0,Y 587.339,Z 400.948,A -85,B 0,C 180,E1 -1301.157,E2 -1301.157} C_VEL
LIN {X 0,Y 587.337,Z 400.948,A -85,B 0,C 180,E1 -1304.114,E2 -1304.114} C_VEL
LIN {X 0,Y 587.315,Z 400.953,A -85,B 0,C 180,E1 -1306.994,E2 -1306.994} C_VEL
LIN {X 0,Y 587.32,Z 400.955,A -85,B 0,C 180,E1 -1309.746,E2 -1309.746} C_VEL
LIN {X 0,Y 587.37,Z 401.12,A -85,B 0,C 180,E1 -1311.819,E2 -1311.819} C_VEL
LIN {X 0,Y 587.568,Z 406.843,A -85,B 0,C 180,E1 -1313.264,E2 -1313.264} C_VEL
LIN {X 0,Y 587.475,Z 418.314,A -85,B 0,C 180,E1 -1316.201,E2 -1316.201} C_VEL
LIN {X 0,Y 587.598,Z 427.801,A -85,B 0,C 180,E1 -1318.649,E2 -1318.649} C_VEL
LIN {X 0,Y 587.602,Z 436.115,A -85,B 0,C 180,E1 -1320.823,E2 -1320.823} C_VEL
LIN {X 0,Y 587.539,Z 446.99,A -85,B 0,C 180,E1 -1323.784,E2 -1323.784} C_VEL
LIN {X 0,Y 587.418,Z 458.153,A -85,B 0,C 180,E1 -1326.745,E2 -1326.745} C_VEL
LIN {X 0,Y 587.381,Z 468.094,A -85,B 0,C 180,E1 -1329.331,E2 -1329.331} C_VEL
LIN {X 0,Y 587.333,Z 479.455,A -85,B 0,C 180,E1 -1332.234,E2 -1332.234} C_VEL
LIN {X 0,Y 587.277,Z 491.651,A -85,B 0,C 180,E1 -1335.299,E2 -1335.299} C_VEL
LIN {X 0,Y 588.008,Z 496.184,A -85,B 0,C 180,E1 -1335.383,E2 -1335.383} C_VEL
LIN {X 0,Y 587.934,Z 510.7,A -85,B 0,C 180,E1 -1335.672,E2 -1335.672} C_VEL
LIN {X 0,Y 587.856,Z 524.952,A -85,B 0,C 180,E1 -1336.106,E2 -1336.106} C_VEL
LIN {X 0,Y 587.772,Z 538.995,A -85,B 0,C 180,E1 -1336.693,E2 -1336.693} C_VEL
LIN {X 0,Y 587.626,Z 551.964,A -85,B 0,C 180,E1 -1337.393,E2 -1337.393} C_VEL
LIN {X 0,Y 587.543,Z 563.726,A -85,B 0,C 180,E1 -1338.18,E2 -1338.18} C_VEL
LIN {X 0,Y 587.467,Z 575.439,A -85,B 0,C 180,E1 -1339.139,E2 -1339.139} C_VEL
LIN {X 0,Y 587.355,Z 585.919,A -85,B 0,C 180,E1 -1340.183,E2 -1340.183} C_VEL
LIN {X 0,Y 587.311,Z 594.571,A -85,B 0,C 180,E1 -1341.224,E2 -1341.224} C_VEL
LIN {X 0,Y 587.25,Z 602.85,A -85,B 0,C 180,E1 -1342.435,E2 -1342.435} C_VEL
LIN {X 0,Y 587.181,Z 609.467,A -85,B 0,C 180,E1 -1343.636,E2 -1343.636} C_VEL
LIN {X 0,Y 587.159,Z 614.789,A -85,B 0,C 180,E1 -1344.85,E2 -1344.85} C_VEL
LIN {X 0,Y 587.181,Z 618.307,A -85,B 0,C 180,E1 -1345.882,E2 -1345.882} C_VEL
LIN {X 0,Y 587.13,Z 621.743,A -85,B 0,C 180,E1 -1347.256,E2 -1347.256} C_VEL
LIN {X 0,Y 587.145,Z 623.786,A -85,B 0,C 180,E1 -1348.628,E2 -1348.628} C_VEL
LIN {X 0,Y 587.136,Z 624.496,A -85,B 0,C 180,E1 -1350,E2 -1350} C_VEL
LIN {X 0,Y 587.142,Z 623.876,A -85,B 0,C 180,E1 -1351.372,E2 -1351.372} C_VEL
LIN {X 0,Y 587.128,Z 621.93,A -85,B 0,C 180,E1 -1352.744,E2 -1352.744} C_VEL
LIN {X 0,Y 587.182,Z 618.584,A -85,B 0,C 180,E1 -1354.118,E2 -1354.118} C_VEL
LIN {X 0,Y 587.2,Z 613.762,A -85,B 0,C 180,E1 -1355.494,E2 -1355.494} C_VEL
LIN {X 0,Y 587.209,Z 608.77,A -85,B 0,C 180,E1 -1356.593,E2 -1356.593} C_VEL
LIN {X 0,Y 587.262,Z 601.217,A -85,B 0,C 180,E1 -1357.91,E2 -1357.91} C_VEL
LIN {X 0,Y 587.332,Z 592.56,A -85,B 0,C 180,E1 -1359.123,E2 -1359.123} C_VEL
LIN {X 0,Y 587.376,Z 583.508,A -85,B 0,C 180,E1 -1360.165,E2 -1360.165} C_VEL
LIN {X 0,Y 587.504,Z 572.537,A -85,B 0,C 180,E1 -1361.209,E2 -1361.209} C_VEL
LIN {X 0,Y 587.578,Z 561.367,A -85,B 0,C 180,E1 -1362.082,E2 -1362.082} C_VEL
LIN {X 0,Y 587.637,Z 549.014,A -85,B 0,C 180,E1 -1362.871,E2 -1362.871} C_VEL
LIN {X 0,Y 587.77,Z 537.152,A -85,B 0,C 180,E1 -1363.483,E2 -1363.483} C_VEL
LIN {X 0,Y 587.872,Z 523.889,A -85,B 0,C 180,E1 -1364.02,E2 -1364.02} C_VEL
LIN {X 0,Y 587.949,Z 510.006,A -85,B 0,C 180,E1 -1364.434,E2 -1364.434} C_VEL
LIN {X 0,Y 587.902,Z 495.07,A -85,B 0,C 180,E1 -1364.726,E2 -1364.726} C_VEL
LIN {X 0,Y 587.242,Z 491.621,A -85,B 0,C 180,E1 -1364.8,E2 -1364.8} C_VEL
LIN {X 0,Y 587.333,Z 479.81,A -85,B 0,C 180,E1 -1367.766,E2 -1367.766} C_VEL
LIN {X 0,Y 587.377,Z 468.443,A -85,B 0,C 180,E1 -1370.669,E2 -1370.669} C_VEL
LIN {X 0,Y 587.417,Z 458.496,A -85,B 0,C 180,E1 -1373.255,E2 -1373.255} C_VEL
LIN {X 0,Y 587.539,Z 447.324,A -85,B 0,C 180,E1 -1376.216,E2 -1376.216} C_VEL
LIN {X 0,Y 587.602,Z 436.441,A -85,B 0,C 180,E1 -1379.177,E2 -1379.177} C_VEL
LIN {X 0,Y 587.577,Z 426.621,A -85,B 0,C 180,E1 -1381.755,E2 -1381.755} C_VEL
LIN {X 0,Y 587.492,Z 415.271,A -85,B 0,C 180,E1 -1384.669,E2 -1384.669} C_VEL
LIN {X 0,Y 587.599,Z 403.806,A -85,B 0,C 180,E1 -1387.589,E2 -1387.589} C_VEL
LIN {X 0,Y 587.347,Z 400.952,A -85,B 0,C 180,E1 -1388.353,E2 -1388.353} C_VEL
LIN {X 0,Y 587.34,Z 400.952,A -85,B 0,C 180,E1 -1391.157,E2 -1391.157} C_VEL
LIN {X 0,Y 587.329,Z 400.951,A -85,B 0,C 180,E1 -1394.113,E2 -1394.113} C_VEL
LIN {X 0,Y 587.327,Z 400.954,A -85,B 0,C 180,E1 -1396.994,E2 -1396.994} C_VEL
LIN {X 0,Y 587.316,Z 400.954,A -85,B 0,C 180,E1 -1399.746,E2 -1399.746} C_VEL
LIN {X 0,Y 587.347,Z 400.949,A -85,B 0,C 180,E1 -1402.392,E2 -1402.392} C_VEL
LIN {X 0,Y 587.328,Z 400.951,A -85,B 0,C 180,E1 -1404.944,E2 -1404.944} C_VEL
LIN {X 0,Y 587.341,Z 400.949,A -85,B 0,C 180,E1 -1407.421,E2 -1407.421} C_VEL
LIN {X 0,Y 587.35,Z 400.947,A -85,B 0,C 180,E1 -1409.831,E2 -1409.831} C_VEL
LIN {X 0,Y 587.354,Z 400.948,A -85,B 0,C 180,E1 -1412.307,E2 -1412.307} C_VEL
LIN {X 0,Y 587.354,Z 400.949,A -85,B 0,C 180,E1 -1415.241,E2 -1415.241} C_VEL
LIN {X 0,Y 587.326,Z 400.951,A -85,B 0,C 180,E1 -1418.226,E2 -1418.226} C_VEL
LIN {X 0,Y 587.354,Z 400.951,A -85,B 0,C 180,E1 -1421.151,E2 -1421.151} C_VEL
LIN {X 0,Y 587.372,Z 400.946,A -85,B 0,C 180,E1 -1423.262,E2 -1423.262} C_VEL
LIN {X 0,Y 588.206,Z 404.687,A -85,B 0,C 180,E1 -1423.381,E2 -1423.381} C_VEL
LIN {X 0,Y 588.107,Z 419.979,A -85,B 0,C 180,E1 -1423.868,E2 -1423.868} C_VEL
LIN {X 0,Y 587.95,Z 434.705,A -85,B 0,C 180,E1 -1424.487,E2 -1424.487} C_VEL
LIN {X 0,Y 587.839,Z 448.013,A -85,B 0,C 180,E1 -1425.194,E2 -1425.194} C_VEL
LIN {X 0,Y 587.734,Z 461.151,A -85,B 0,C 180,E1 -1426.048,E2 -1426.048} C_VEL
LIN {X 0,Y 587.565,Z 472.787,A -85,B 0,C 180,E1 -1426.952,E2 -1426.952} C_VEL
LIN {X 0,Y 587.472,Z 485.068,A -85,B 0,C 180,E1 -1428.091,E2 -1428.091} C_VEL
LIN {X 0,Y 587.384,Z 495.924,A -85,B 0,C 180,E1 -1429.312,E2 -1429.312} C_VEL
LIN {X 0,Y 587.285,Z 504.985,A -85,B 0,C 180,E1 -1430.529,E2 -1430.529} C_VEL
LIN {X 0,Y 587.254,Z 512.496,A -85,B 0,C 180,E1 -1431.743,E2 -1431.743} C_VEL
LIN {X 0,Y 587.208,Z 519.502,A -85,B 0,C 180,E1 -1433.126,E2 -1433.126} C_VEL
LIN {X 0,Y 587.196,Z 524.99,A -85,B 0,C 180,E1 -1434.505,E2 -1434.505} C_VEL
LIN {X 0,Y 587.167,Z 529.177,A -85,B 0,C 180,E1 -1435.882,E2 -1435.882} C_VEL
LIN {X 0,Y 587.128,Z 532.12,A -85,B 0,C 180,E1 -1437.256,E2 -1437.256} C_VEL
LIN {X 0,Y 587.142,Z 533.875,A -85,B 0,C 180,E1 -1438.628,E2 -1438.628} C_VEL
LIN {X 0,Y 587.135,Z 534.484,A -85,B 0,C 180,E1 -1440,E2 -1440} C_VEL
LIN {X 0,Y 587.147,Z 533.938,A -85,B 0,C 180,E1 -1441.372,E2 -1441.372} C_VEL
LIN {X 0,Y 587.13,Z 532.257,A -85,B 0,C 180,E1 -1442.744,E2 -1442.744} C_VEL
LIN {X 0,Y 587.167,Z 529.413,A -85,B 0,C 180,E1 -1444.118,E2 -1444.118} C_VEL
LIN {X 0,Y 587.199,Z 525.322,A -85,B 0,C 180,E1 -1445.494,E2 -1445.494} C_VEL
LIN {X 0,Y 587.208,Z 519.896,A -85,B 0,C 180,E1 -1446.874,E2 -1446.874} C_VEL
LIN {X 0,Y 587.251,Z 513.003,A -85,B 0,C 180,E1 -1448.257,E2 -1448.257} C_VEL
LIN {X 0,Y 587.287,Z 504.409,A -85,B 0,C 180,E1 -1449.645,E2 -1449.645} C_VEL
LIN {X 0,Y 587.347,Z 495.235,A -85,B 0,C 180,E1 -1450.863,E2 -1450.863} C_VEL
LIN {X 0,Y 587.447,Z 485.906,A -85,B 0,C 180,E1 -1451.91,E2 -1451.91} C_VEL
LIN {X 0,Y 587.558,Z 474.883,A -85,B 0,C 180,E1 -1452.96,E2 -1452.96} C_VEL
LIN {X 0,Y 587.711,Z 462.429,A -85,B 0,C 180,E1 -1453.953,E2 -1453.953} C_VEL
LIN {X 0,Y 587.823,Z 449.481,A -85,B 0,C 180,E1 -1454.807,E2 -1454.807} C_VEL
LIN {X 0,Y 587.94,Z 436.474,A -85,B 0,C 180,E1 -1455.513,E2 -1455.513} C_VEL
LIN {X 0,Y 588.086,Z 422.352,A -85,B 0,C 180,E1 -1456.132,E2 -1456.132} C_VEL
LIN {X 0,Y 588.188,Z 407.808,A -85,B 0,C 180,E1 -1456.62,E2 -1456.62} C_VEL
LIN {X 0,Y 588.055,Z 403.408,A -85,B 0,C 180,E1 -1456.745,E2 -1456.745} C_VEL
LIN {X 0,Y 587.376,Z 400.941,A -85,B 0,C 180,E1 -1456.837,E2 -1456.837} C_VEL
LIN {X 0,Y 587.346,Z 400.946,A -85,B 0,C 180,E1 -1459.575,E2 -1459.575} C_VEL
LIN {X 0,Y 587.343,Z 400.945,A -85,B 0,C 180,E1 -1462.514,E2 -1462.514} C_VEL
LIN {X 0,Y 587.354,Z 400.942,A -85,B 0,C 180,E1 -1464.758,E2 -1464.758} C_VEL
LIN {X 0,Y 587.331,Z 400.945,A -85,B 0,C 180,E1 -1467.046,E2 -1467.046} C_VEL
LIN {X 0,Y 587.35,Z 400.945,A -85,B 0,C 180,E1 -1469.379,E2 -1469.379} C_VEL
LIN {X 0,Y 587.359,Z 400.95,A -85,B 0,C 180,E1 -1471.838,E2 -1471.838} C_VEL
LIN {X 0,Y 587.349,Z 400.944,A -85,B 0,C 180,E1 -1474.348,E2 -1474.348} C_VEL
LIN {X 0,Y 587.346,Z 400.952,A -85,B 0,C 180,E1 -1477.608,E2 -1477.608} C_VEL
LIN {X 0,Y 587.314,Z 400.948,A -85,B 0,C 180,E1 -1480.254,E2 -1480.254} C_VEL
LIN {X 0,Y 587.324,Z 400.948,A -85,B 0,C 180,E1 -1483.006,E2 -1483.006} C_VEL
LIN {X 0,Y 587.306,Z 401.067,A -85,B 0,C 180,E1 -1485.142,E2 -1485.142} C_VEL
LIN {X 0,Y 587.288,Z 414.738,A -85,B 0,C 180,E1 -1488.382,E2 -1488.382} C_VEL
LIN {X 0,Y 587.623,Z 424.155,A -85,B 0,C 180,E1 -1490.663,E2 -1490.663} C_VEL
LIN {X 0,Y 587.725,Z 427.236,A -85,B 0,C 180,E1 -1491.551,E2 -1491.551} C_VEL
LIN {X 0,Y 587.645,Z 435.42,A -85,B 0,C 180,E1 -1494.415,E2 -1494.415} C_VEL
LIN {X 0,Y 587.59,Z 442.612,A -85,B 0,C 180,E1 -1496.851,E2 -1496.851} C_VEL
LIN {X 0,Y 587.499,Z 451.711,A -85,B 0,C 180,E1 -1499.839,E2 -1499.839} C_VEL
LIN {X 0,Y 587.469,Z 459.36,A -85,B 0,C 180,E1 -1502.286,E2 -1502.286} C_VEL
LIN {X 0,Y 587.412,Z 467.62,A -85,B 0,C 180,E1 -1504.866,E2 -1504.866} C_VEL
LIN {X 0,Y 587.36,Z 476.186,A -85,B 0,C 180,E1 -1507.487,E2 -1507.487} C_VEL
LIN {X 0,Y 587.324,Z 485.976,A -85,B 0,C 180,E1 -1510.424,E2 -1510.424} C_VEL
LIN {X 0,Y 587.278,Z 495.766,A -85,B 0,C 180,E1 -1513.309,E2 -1513.309} C_VEL
LIN {X 0,Y 587.255,Z 502.473,A -85,B 0,C 180,E1 -1515.26,E2 -1515.26} C_VEL
LIN {X 0,Y 588.023,Z 508.429,A -85,B 0,C 180,E1 -1515.372,E2 -1515.372} C_VEL
LIN {X 0,Y 587.915,Z 522.733,A -85,B 0,C 180,E1 -1515.679,E2 -1515.679} C_VEL
LIN {X 0,Y 587.861,Z 536.117,A -85,B 0,C 180,E1 -1516.104,E2 -1516.104} C_VEL
LIN {X 0,Y 587.744,Z 549.893,A -85,B 0,C 180,E1 -1516.692,E2 -1516.692} C_VEL
LIN {X 0,Y 587.624,Z 562.69,A -85,B 0,C 180,E1 -1517.393,E2 -1517.393} C_VEL
LIN {X 0,Y 587.513,Z 575.479,A -85,B 0,C 180,E1 -1518.267,E2 -1518.267} C_VEL
LIN {X 0,Y 587.465,Z 585.938,A -85,B 0,C 180,E1 -1519.139,E2 -1519.139} C_VEL
LIN {X 0,Y 587.353,Z 596.331,A -85,B 0,C 180,E1 -1520.183,E2 -1520.183} C_VEL
LIN {X 0,Y 587.311,Z 604.908,A -85,B 0,C 180,E1 -1521.224,E2 -1521.224} C_VEL
LIN {X 0,Y 587.249,Z 613.118,A -85,B 0,C 180,E1 -1522.435,E2 -1522.435} C_VEL
LIN {X 0,Y 587.18,Z 619.685,A -85,B 0,C 180,E1 -1523.635,E2 -1523.635} C_VEL
LIN {X 0,Y 587.16,Z 624.964,A -85,B 0,C 180,E1 -1524.85,E2 -1524.85} C_VEL
LIN {X 0,Y 587.179,Z 628.444,A -85,B 0,C 180,E1 -1525.882,E2 -1525.882} C_VEL
LIN {X 0,Y 587.13,Z 631.832,A -85,B 0,C 180,E1 -1527.256,E2 -1527.256} C_VEL
LIN {X 0,Y 587.141,Z 633.83,A -85,B 0,C 180,E1 -1528.628,E2 -1528.628} C_VEL
LIN {X 0,Y 587.135,Z 634.5,A -85,B 0,C 180,E1 -1530,E2 -1530} C_VEL
LIN {X 0,Y 587.141,Z 633.831,A -85,B 0,C 180,E1 -1531.372,E2 -1531.372} C_VEL
LIN {X 0,Y 587.13,Z 631.834,A -85,B 0,C 180,E1 -1532.744,E2 -1532.744} C_VEL
LIN {X 0,Y 587.179,Z 628.446,A -85,B 0,C 180,E1 -1534.118,E2 -1534.118} C_VEL
LIN {X 0,Y 587.199,Z 623.573,A -85,B 0,C 180,E1 -1535.494,E2 -1535.494} C_VEL
LIN {X 0,Y 587.209,Z 617.057,A -85,B 0,C 180,E1 -1536.874,E2 -1536.874} C_VEL
LIN {X 0,Y 587.268,Z 609.802,A -85,B 0,C 180,E1 -1538.083,E2 -1538.083} C_VEL
LIN {X 0,Y 587.321,Z 600.823,A -85,B 0,C 180,E1 -1539.297,E2 -1539.297} C_VEL
LIN {X 0,Y 587.372,Z 591.391,A -85,B 0,C 180,E1 -1540.339,E2 -1540.339} C_VEL
LIN {X 0,Y 587.475,Z 581.022,A -85,B 0,C 180,E1 -1541.29,E2 -1541.29} C_VEL
LIN {X 0,Y 587.578,Z 569.427,A -85,B 0,C 180,E1 -1542.17,E2 -1542.17} C_VEL
LIN {X 0,Y 587.651,Z 556.65,A -85,B 0,C 180,E1 -1542.958,E2 -1542.958} C_VEL
LIN {X 0,Y 587.799,Z 543.184,A -85,B 0,C 180,E1 -1543.615,E2 -1543.615} C_VEL
LIN {X 0,Y 587.904,Z 528.856,A -85,B 0,C 180,E1 -1544.143,E2 -1544.143} C_VEL
LIN {X 0,Y 587.983,Z 514.834,A -85,B 0,C 180,E1 -1544.508,E2 -1544.508} C_VEL
LIN {X 0,Y 587.832,Z 505.675,A -85,B 0,C 180,E1 -1544.673,E2 -1544.673} C_VEL
LIN {X 0,Y 587.264,Z 502.46,A -85,B 0,C 180,E1 -1544.743,E2 -1544.743} C_VEL
LIN {X 0,Y 587.302,Z 492.095,A -85,B 0,C 180,E1 -1547.767,E2 -1547.767} C_VEL
LIN {X 0,Y 587.343,Z 482.305,A -85,B 0,C 180,E1 -1550.67,E2 -1550.67} C_VEL
LIN {X 0,Y 587.381,Z 472.515,A -85,B 0,C 180,E1 -1553.63,E2 -1553.63} C_VEL
LIN {X 0,Y 587.445,Z 463.949,A -85,B 0,C 180,E1 -1556.274,E2 -1556.274} C_VEL
LIN {X 0,Y 587.519,Z 454.805,A -85,B 0,C 180,E1 -1559.163,E2 -1559.163} C_VEL
LIN {X 0,Y 587.549,Z 446.479,A -85,B 0,C 180,E1 -1561.868,E2 -1561.868} C_VEL
LIN {X 0,Y 587.659,Z 438.909,A -85,B 0,C 180,E1 -1564.392,E2 -1564.392} C_VEL
LIN {X 0,Y 587.682,Z 430.908,A -85,B 0,C 180,E1 -1567.151,E2 -1567.151} C_VEL
LIN {X 0,Y 587.682,Z 424.553,A -85,B 0,C 180,E1 -1569.332,E2 -1569.332} C_VEL
LIN {X 0,Y 587.645,Z 416.193,A -85,B 0,C 180,E1 -1572.141,E2 -1572.141} C_VEL
LIN {X 0,Y 587.745,Z 408.442,A -85,B 0,C 180,E1 -1574.87,E2 -1574.87} C_VEL
LIN {X 0,Y 587.702,Z 403.079,A -85,B 0,C 180,E1 -1576.842,E2 -1576.842} C_VEL
LIN {X 0,Y 587.334,Z 400.951,A -85,B 0,C 180,E1 -1577.695,E2 -1577.695} C_VEL
LIN {X 0,Y 587.332,Z 400.952,A -85,B 0,C 180,E1 -1580.64,E2 -1580.64} C_VEL
LIN {X 0,Y 587.355,Z 400.946,A -85,B 0,C 180,E1 -1583.292,E2 -1583.292} C_VEL
LIN {X 0,Y 587.365,Z 400.945,A -85,B 0,C 180,E1 -1585.78,E2 -1585.78} C_VEL
LIN {X 0,Y 587.345,Z 400.95,A -85,B 0,C 180,E1 -1588.231,E2 -1588.231} C_VEL
LIN {X 0,Y 587.353,Z 400.946,A -85,B 0,C 180,E1 -1590.866,E2 -1590.866} C_VEL
LIN {X 0,Y 587.362,Z 400.943,A -85,B 0,C 180,E1 -1593.819,E2 -1593.819} C_VEL
LIN {X 0,Y 587.342,Z 400.952,A -85,B 0,C 180,E1 -1595.994,E2 -1595.994} C_VEL
LIN {X 0,Y 587.325,Z 400.948,A -85,B 0,C 180,E1 -1598.226,E2 -1598.226} C_VEL
LIN {X 0,Y 587.351,Z 400.945,A -85,B 0,C 180,E1 -1601.151,E2 -1601.151} C_VEL
LIN {X 0,Y 587.356,Z 400.949,A -85,B 0,C 180,E1 -1603.311,E2 -1603.311} C_VEL
LIN {X 0,Y 587.359,Z 400.946,A -85,B 0,C 180,E1 -1606.154,E2 -1606.154} C_VEL
LIN {X 0,Y 587.344,Z 400.947,A -85,B 0,C 180,E1 -1608.963,E2 -1608.963} C_VEL
LIN {X 0,Y 587.344,Z 400.945,A -85,B 0,C 180,E1 -1611.744,E2 -1611.744} C_VEL
LIN {X 0,Y 587.36,Z 400.945,A -85,B 0,C 180,E1 -1614.507,E2 -1614.507} C_VEL
LIN {X 0,Y 587.379,Z 400.943,A -85,B 0,C 180,E1 -1617.257,E2 -1617.257} C_VEL
LIN {X 0,Y 587.384,Z 400.948,A -85,B 0,C 180,E1 -1620,E2 -1620} C_VEL
LIN {X 0,Y 587.38,Z 400.944,A -85,B 0,C 180,E1 -1622.743,E2 -1622.743} C_VEL
LIN {X 0,Y 587.357,Z 400.945,A -85,B 0,C 180,E1 -1625.493,E2 -1625.493} C_VEL
LIN {X 0,Y 587.371,Z 400.942,A -85,B 0,C 180,E1 -1628.255,E2 -1628.255} C_VEL
LIN {X 0,Y 587.351,Z 400.946,A -85,B 0,C 180,E1 -1631.134,E2 -1631.134} C_VEL
LIN {X 0,Y 587.368,Z 400.943,A -85,B 0,C 180,E1 -1634.26,E2 -1634.26} C_VEL
LIN {X 0,Y 587.352,Z 400.945,A -85,B 0,C 180,E1 -1637.406,E2 -1637.406} C_VEL
LIN {X 0,Y 587.312,Z 400.952,A -85,B 0,C 180,E1 -1638.313,E2 -1638.313} C_VEL
LIN {X 0,Y 586.669,Z 401.03,A -85,B 0,C 180,E1 -1638.886,E2 -1638.886} C_VEL
LIN {X 0,Y 583.844,Z 401.385,A -85,B 0,C 180,E1 -1639.814,E2 -1639.814} C_VEL
LIN {X 0,Y 581.434,Z 401.688,A -85,B 0,C 180,E1 -1640.561,E2 -1640.561} C_VEL
LIN {X 0,Y 580.381,Z 401.819,A -85,B 0,C 180,E1 -1641.138,E2 -1641.138} C_VEL
LIN {X 0,Y 580.286,Z 401.828,A -85,B 0,C 180,E1 -1641.333,E2 -1641.333} C_VEL
LIN {X 0,Y 580.302,Z 401.827,A -85,B 0,C 180,E1 -1644.316,E2 -1644.316} C_VEL
LIN {X 0,Y 580.283,Z 401.826,A -85,B 0,C 180,E1 -1646.623,E2 -1646.623} C_VEL
LIN {X 0,Y 580.304,Z 401.823,A -85,B 0,C 180,E1 -1649.31,E2 -1649.31} C_VEL
LIN {X 0,Y 580.304,Z 401.824,A -85,B 0,C 180,E1 -1652.2,E2 -1652.2} C_VEL
LIN {X 0,Y 580.291,Z 401.83,A -85,B 0,C 180,E1 -1654.696,E2 -1654.696} C_VEL
LIN {X 0,Y 580.301,Z 401.826,A -85,B 0,C 180,E1 -1657.268,E2 -1657.268} C_VEL
LIN {X 0,Y 580.295,Z 401.826,A -85,B 0,C 180,E1 -1660.271,E2 -1660.271} C_VEL
LIN {X 0,Y 580.284,Z 401.827,A -85,B 0,C 180,E1 -1662.706,E2 -1662.706} C_VEL
LIN {X 0,Y 580.273,Z 401.829,A -85,B 0,C 180,E1 -1665.609,E2 -1665.609} C_VEL
LIN {X 0,Y 580.282,Z 401.833,A -85,B 0,C 180,E1 -1668.231,E2 -1668.231} C_VEL
LIN {X 0,Y 580.292,Z 401.83,A -85,B 0,C 180,E1 -1670.966,E2 -1670.966} C_VEL
LIN {X 0,Y 580.333,Z 402.04,A -85,B 0,C 180,E1 -1671.691,E2 -1671.691} C_VEL
LIN {X 0,Y 580.634,Z 406.246,A -85,B 0,C 180,E1 -1672.757,E2 -1672.757} C_VEL
LIN {X 0,Y 580.484,Z 417.951,A -85,B 0,C 180,E1 -1675.784,E2 -1675.784} C_VEL
LIN {X 0,Y 580.606,Z 428.889,A -85,B 0,C 180,E1 -1678.634,E2 -1678.634} C_VEL
LIN {X 0,Y 580.609,Z 439.69,A -85,B 0,C 180,E1 -1681.437,E2 -1681.437} C_VEL
LIN {X 0,Y 580.538,Z 449.635,A -85,B 0,C 180,E1 -1684.163,E2 -1684.163} C_VEL
LIN {X 0,Y 580.431,Z 460.996,A -85,B 0,C 180,E1 -1687.203,E2 -1687.203} C_VEL
LIN {X 0,Y 580.322,Z 470.936,A -85,B 0,C 180,E1 -1689.809,E2 -1689.809} C_VEL
LIN {X 0,Y 580.28,Z 482.298,A -85,B 0,C 180,E1 -1692.739,E2 -1692.739} C_VEL
LIN {X 0,Y 580.224,Z 491.709,A -85,B 0,C 180,E1 -1695.118,E2 -1695.118} C_VEL
LIN {X 0,Y 581.155,Z 497.205,A -85,B 0,C 180,E1 -1695.221,E2 -1695.221} C_VEL
LIN {X 0,Y 581.054,Z 511.896,A -85,B 0,C 180,E1 -1695.529,E2 -1695.529} C_VEL
LIN {X 0,Y 580.972,Z 525.114,A -85,B 0,C 180,E1 -1695.943,E2 -1695.943} C_VEL
LIN {X 0,Y 580.835,Z 539.006,A -85,B 0,C 180,E1 -1696.531,E2 -1696.531} C_VEL
LIN {X 0,Y 580.689,Z 551.972,A -85,B 0,C 180,E1 -1697.239,E2 -1697.239} C_VEL
LIN {X 0,Y 580.564,Z 563.737,A -85,B 0,C 180,E1 -1698.035,E2 -1698.035} C_VEL
LIN {X 0,Y 580.463,Z 575.459,A -85,B 0,C 180,E1 -1699.008,E2 -1699.008} C_VEL
LIN {X 0,Y 580.318,Z 585.926,A -85,B 0,C 180,E1 -1700.062,E2 -1700.062} C_VEL
LIN {X 0,Y 580.254,Z 594.574,A -85,B 0,C 180,E1 -1701.116,E2 -1701.116} C_VEL
LIN {X 0,Y 580.177,Z 602.853,A -85,B 0,C 180,E1 -1702.343,E2 -1702.343} C_VEL
LIN {X 0,Y 580.124,Z 608.765,A -85,B 0,C 180,E1 -1703.416,E2 -1703.416} C_VEL
LIN {X 0,Y 580.128,Z 613.395,A -85,B 0,C 180,E1 -1704.438,E2 -1704.438} C_VEL
LIN {X 0,Y 580.104,Z 618.311,A -85,B 0,C 180,E1 -1705.831,E2 -1705.831} C_VEL
LIN {X 0,Y 580.041,Z 621.746,A -85,B 0,C 180,E1 -1707.222,E2 -1707.222} C_VEL
LIN {X 0,Y 580.045,Z 623.787,A -85,B 0,C 180,E1 -1708.611,E2 -1708.611} C_VEL
LIN {X 0,Y 580.037,Z 624.496,A -85,B 0,C 180,E1 -1710,E2 -1710} C_VEL
LIN {X 0,Y 580.042,Z 623.874,A -85,B 0,C 180,E1 -1711.389,E2 -1711.389} C_VEL
LIN {X 0,Y 580.039,Z 621.93,A -85,B 0,C 180,E1 -1712.778,E2 -1712.778} C_VEL
LIN {X 0,Y 580.105,Z 618.583,A -85,B 0,C 180,E1 -1714.169,E2 -1714.169} C_VEL
LIN {X 0,Y 580.129,Z 613.762,A -85,B 0,C 180,E1 -1715.562,E2 -1715.562} C_VEL
LIN {X 0,Y 580.142,Z 607.291,A -85,B 0,C 180,E1 -1716.958,E2 -1716.958} C_VEL
LIN {X 0,Y 580.193,Z 600.095,A -85,B 0,C 180,E1 -1718.183,E2 -1718.183} C_VEL
LIN {X 0,Y 580.275,Z 591.177,A -85,B 0,C 180,E1 -1719.41,E2 -1719.41} C_VEL
LIN {X 0,Y 580.356,Z 581.844,A -85,B 0,C 180,E1 -1720.466,E2 -1720.466} C_VEL
LIN {X 0,Y 580.465,Z 570.441,A -85,B 0,C 180,E1 -1721.523,E2 -1721.523} C_VEL
LIN {X 0,Y 580.603,Z 558.811,A -85,B 0,C 180,E1 -1722.407,E2 -1722.407} C_VEL
LIN {X 0,Y 580.733,Z 545.874,A -85,B 0,C 180,E1 -1723.204,E2 -1723.204} C_VEL
LIN {X 0,Y 580.892,Z 533.203,A -85,B 0,C 180,E1 -1723.824,E2 -1723.824} C_VEL
LIN {X 0,Y 581.004,Z 519.034,A -85,B 0,C 180,E1 -1724.353,E2 -1724.353} C_VEL
LIN {X 0,Y 581.126,Z 504.512,A -85,B 0,C 180,E1 -1724.735,E2 -1724.735} C_VEL
LIN {X 0,Y 580.977,Z 495.726,A -85,B 0,C 180,E1 -1724.896,E2 -1724.896} C_VEL
LIN {X 0,Y 580.221,Z 491.619,A -85,B 0,C 180,E1 -1724.983,E2 -1724.983} C_VEL
LIN {X 0,Y 580.283,Z 479.808,A -85,B 0,C 180,E1 -1727.989,E2 -1727.989} C_VEL
LIN {X 0,Y 580.346,Z 468.663,A -85,B 0,C 180,E1 -1730.873,E2 -1730.873} C_VEL
LIN {X 0,Y 580.41,Z 458.493,A -85,B 0,C 180,E1 -1733.552,E2 -1733.552} C_VEL
LIN {X 0,Y 580.554,Z 447.947,A -85,B 0,C 180,E1 -1736.386,E2 -1736.386} C_VEL
LIN {X 0,Y 580.623,Z 438.526,A -85,B 0,C 180,E1 -1738.958,E2 -1738.958} C_VEL
LIN {X 0,Y 580.573,Z 427.883,A -85,B 0,C 180,E1 -1741.718,E2 -1741.718} C_VEL
LIN {X 0,Y 580.513,Z 416.863,A -85,B 0,C 180,E1 -1744.589,E2 -1744.589} C_VEL
LIN {X 0,Y 580.621,Z 406.587,A -85,B 0,C 180,E1 -1747.244,E2 -1747.244} C_VEL
LIN {X 0,Y 580.297,Z 401.83,A -85,B 0,C 180,E1 -1748.477,E2 -1748.477} C_VEL
LIN {X 0,Y 580.286,Z 401.829,A -85,B 0,C 180,E1 -1751.332,E2 -1751.332} C_VEL
LIN {X 0,Y 580.281,Z 401.83,A -85,B 0,C 180,E1 -1753.658,E2 -1753.658} C_VEL
LIN {X 0,Y 580.289,Z 401.828,A -85,B 0,C 180,E1 -1756.608,E2 -1756.608} C_VEL
LIN {X 0,Y 580.301,Z 401.828,A -85,B 0,C 180,E1 -1759.157,E2 -1759.157} C_VEL
LIN {X 0,Y 580.291,Z 401.831,A -85,B 0,C 180,E1 -1761.927,E2 -1761.927} C_VEL
LIN {X 0,Y 580.288,Z 401.829,A -85,B 0,C 180,E1 -1764.455,E2 -1764.455} C_VEL
LIN {X 0,Y 580.293,Z 401.828,A -85,B 0,C 180,E1 -1766.975,E2 -1766.975} C_VEL
LIN {X 0,Y 580.31,Z 401.824,A -85,B 0,C 180,E1 -1769.426,E2 -1769.426} C_VEL
LIN {X 0,Y 580.301,Z 401.826,A -85,B 0,C 180,E1 -1772.141,E2 -1772.141} C_VEL
LIN {X 0,Y 580.324,Z 401.825,A -85,B 0,C 180,E1 -1775.27,E2 -1775.27} C_VEL
LIN {X 0,Y 580.276,Z 401.829,A -85,B 0,C 180,E1 -1777.947,E2 -1777.947} C_VEL
LIN {X 0,Y 580.322,Z 401.826,A -85,B 0,C 180,E1 -1780.914,E2 -1780.914} C_VEL
LIN {X 0,Y 580.336,Z 401.938,A -85,B 0,C 180,E1 -1783.079,E2 -1783.079} C_VEL
LIN {X 0,Y 581.388,Z 406.289,A -85,B 0,C 180,E1 -1783.225,E2 -1783.225} C_VEL
LIN {X 0,Y 581.26,Z 421.18,A -85,B 0,C 180,E1 -1783.718,E2 -1783.718} C_VEL
LIN {X 0,Y 581.068,Z 436.499,A -85,B 0,C 180,E1 -1784.388,E2 -1784.388} C_VEL
LIN {X 0,Y 580.923,Z 449.453,A -85,B 0,C 180,E1 -1785.103,E2 -1785.103} C_VEL
LIN {X 0,Y 580.8,Z 461.319,A -85,B 0,C 180,E1 -1785.89,E2 -1785.89} C_VEL
LIN {X 0,Y 580.599,Z 472.791,A -85,B 0,C 180,E1 -1786.792,E2 -1786.792} C_VEL
LIN {X 0,Y 580.47,Z 485.071,A -85,B 0,C 180,E1 -1787.945,E2 -1787.945} C_VEL
LIN {X 0,Y 580.333,Z 495.116,A -85,B 0,C 180,E1 -1789.08,E2 -1789.08} C_VEL
LIN {X 0,Y 580.234,Z 503.755,A -85,B 0,C 180,E1 -1790.237,E2 -1790.237} C_VEL
LIN {X 0,Y 580.184,Z 511.49,A -85,B 0,C 180,E1 -1791.466,E2 -1791.466} C_VEL
LIN {X 0,Y 580.131,Z 517.892,A -85,B 0,C 180,E1 -1792.692,E2 -1792.692} C_VEL
LIN {X 0,Y 580.129,Z 523.753,A -85,B 0,C 180,E1 -1794.089,E2 -1794.089} C_VEL
LIN {X 0,Y 580.042,Z 527.257,A -85,B 0,C 180,E1 -1795.135,E2 -1795.135} C_VEL
LIN {X 0,Y 580.106,Z 530.781,A -85,B 0,C 180,E1 -1796.527,E2 -1796.527} C_VEL
LIN {X 0,Y 580.034,Z 533.141,A -85,B 0,C 180,E1 -1797.917,E2 -1797.917} C_VEL
LIN {X 0,Y 580.034,Z 534.327,A -85,B 0,C 180,E1 -1799.306,E2 -1799.306} C_VEL
LIN {X 0,Y 580.038,Z 534.364,A -85,B 0,C 180,E1 -1800.694,E2 -1800.694} C_VEL
LIN {X 0,Y 580.037,Z 533.254,A -85,B 0,C 180,E1 -1802.083,E2 -1802.083} C_VEL
LIN {X 0,Y 580.108,Z 530.978,A -85,B 0,C 180,E1 -1803.473,E2 -1803.473} C_VEL
LIN {X 0,Y 580.04,Z 527.519,A -85,B 0,C 180,E1 -1804.865,E2 -1804.865} C_VEL
LIN {X 0,Y 580.094,Z 522.8,A -85,B 0,C 180,E1 -1806.26,E2 -1806.26} C_VEL
LIN {X 0,Y 580.157,Z 516.657,A -85,B 0,C 180,E1 -1807.658,E2 -1807.658} C_VEL
LIN {X 0,Y 580.207,Z 508.91,A -85,B 0,C 180,E1 -1809.06,E2 -1809.06} C_VEL
LIN {X 0,Y 580.288,Z 500.664,A -85,B 0,C 180,E1 -1810.291,E2 -1810.291} C_VEL
LIN {X 0,Y 580.384,Z 490.791,A -85,B 0,C 180,E1 -1811.525,E2 -1811.525} C_VEL
LIN {X 0,Y 580.513,Z 480.651,A -85,B 0,C 180,E1 -1812.587,E2 -1812.587} C_VEL
LIN {X 0,Y 580.652,Z 469.625,A -85,B 0,C 180,E1 -1813.563,E2 -1813.563} C_VEL
LIN {X 0,Y 580.772,Z 458.174,A -85,B 0,C 180,E1 -1814.422,E2 -1814.422} C_VEL
LIN {X 0,Y 580.973,Z 444.911,A -85,B 0,C 180,E1 -1815.255,E2 -1815.255} C_VEL
LIN {X 0,Y 581.156,Z 429.836,A -85,B 0,C 180,E1 -1816.014,E2 -1816.014} C_VEL
LIN {X 0,Y 581.302,Z 414.957,A -85,B 0,C 180,E1 -1816.596,E2 -1816.596} C_VEL
LIN {X 0,Y 581.29,Z 405.082,A -85,B 0,C 180,E1 -1816.903,E2 -1816.903} C_VEL
LIN {X 0,Y 580.328,Z 401.819,A -85,B 0,C 180,E1 -1817.023,E2 -1817.023} C_VEL
LIN {X 0,Y 580.308,Z 401.826,A -85,B 0,C 180,E1 -1819.822,E2 -1819.822} C_VEL
LIN {X 0,Y 580.297,Z 401.821,A -85,B 0,C 180,E1 -1822.802,E2 -1822.802} C_VEL
LIN {X 0,Y 580.31,Z 401.82,A -85,B 0,C 180,E1 -1825.08,E2 -1825.08} C_VEL
LIN {X 0,Y 580.304,Z 401.825,A -85,B 0,C 180,E1 -1828.185,E2 -1828.185} C_VEL
LIN {X 0,Y 580.294,Z 401.821,A -85,B 0,C 180,E1 -1830.696,E2 -1830.696} C_VEL
LIN {X 0,Y 580.307,Z 401.823,A -85,B 0,C 180,E1 -1833.317,E2 -1833.317} C_VEL
LIN {X 0,Y 580.249,Z 401.836,A -85,B 0,C 180,E1 -1835.756,E2 -1835.756} C_VEL
LIN {X 0,Y 580.289,Z 401.824,A -85,B 0,C 180,E1 -1838.146,E2 -1838.146} C_VEL
LIN {X 0,Y 580.3,Z 401.821,A -85,B 0,C 180,E1 -1840.843,E2 -1840.843} C_VEL
LIN {X 0,Y 580.29,Z 401.83,A -85,B 0,C 180,E1 -1843.657,E2 -1843.657} C_VEL
LIN {X 0,Y 580.277,Z 401.875,A -85,B 0,C 180,E1 -1845.131,E2 -1845.131} C_VEL
LIN {X 0,Y 580.213,Z 414.658,A -85,B 0,C 180,E1 -1848.225,E2 -1848.225} C_VEL
LIN {X 0,Y 580.598,Z 425.941,A -85,B 0,C 180,E1 -1850.991,E2 -1850.991} C_VEL
LIN {X 0,Y 580.752,Z 429.486,A -85,B 0,C 180,E1 -1851.89,E2 -1851.89} C_VEL
LIN {X 0,Y 580.696,Z 437.026,A -85,B 0,C 180,E1 -1854.484,E2 -1854.484} C_VEL
LIN {X 0,Y 580.601,Z 444.369,A -85,B 0,C 180,E1 -1856.995,E2 -1856.995} C_VEL
LIN {X 0,Y 580.496,Z 452.935,A -85,B 0,C 180,E1 -1859.839,E2 -1859.839} C_VEL
LIN {X 0,Y 580.487,Z 459.932,A -85,B 0,C 180,E1 -1862.106,E2 -1862.106} C_VEL
LIN {X 0,Y 580.377,Z 468.844,A -85,B 0,C 180,E1 -1864.923,E2 -1864.923} C_VEL
LIN {X 0,Y 580.321,Z 477.41,A -85,B 0,C 180,E1 -1867.574,E2 -1867.574} C_VEL
LIN {X 0,Y 580.268,Z 485.976,A -85,B 0,C 180,E1 -1870.176,E2 -1870.176} C_VEL
LIN {X 0,Y 580.23,Z 495.812,A -85,B 0,C 180,E1 -1873.114,E2 -1873.114} C_VEL
LIN {X 0,Y 580.188,Z 502.599,A -85,B 0,C 180,E1 -1875.084,E2 -1875.084} C_VEL
LIN {X 0,Y 581.159,Z 508.65,A -85,B 0,C 180,E1 -1875.199,E2 -1875.199} C_VEL
LIN {X 0,Y 581.046,Z 522.937,A -85,B 0,C 180,E1 -1875.512,E2 -1875.512} C_VEL
LIN {X 0,Y 580.974,Z 536.246,A -85,B 0,C 180,E1 -1875.941,E2 -1875.941} C_VEL
LIN {X 0,Y 580.837,Z 549.897,A -85,B 0,C 180,E1 -1876.531,E2 -1876.531} C_VEL
LIN {X 0,Y 580.665,Z 562.693,A -85,B 0,C 180,E1 -1877.239,E2 -1877.239} C_VEL
LIN {X 0,Y 580.544,Z 575.481,A -85,B 0,C 180,E1 -1878.124,E2 -1878.124} C_VEL
LIN {X 0,Y 580.461,Z 585.971,A -85,B 0,C 180,E1 -1879.009,E2 -1879.009} C_VEL
LIN {X 0,Y 580.311,Z 596.329,A -85,B 0,C 180,E1 -1880.062,E2 -1880.062} C_VEL
LIN {X 0,Y 580.254,Z 604.906,A -85,B 0,C 180,E1 -1881.116,E2 -1881.116} C_VEL
LIN {X 0,Y 580.176,Z 613.119,A -85,B 0,C 180,E1 -1882.343,E2 -1882.343} C_VEL
LIN {X 0,Y 580.123,Z 618.989,A -85,B 0,C 180,E1 -1883.416,E2 -1883.416} C_VEL
LIN {X 0,Y 580.128,Z 623.572,A -85,B 0,C 180,E1 -1884.438,E2 -1884.438} C_VEL
LIN {X 0,Y 580.102,Z 628.445,A -85,B 0,C 180,E1 -1885.831,E2 -1885.831} C_VEL
LIN {X 0,Y 580.041,Z 631.832,A -85,B 0,C 180,E1 -1887.222,E2 -1887.222} C_VEL
LIN {X 0,Y 580.041,Z 633.83,A -85,B 0,C 180,E1 -1888.611,E2 -1888.611} C_VEL
LIN {X 0,Y 580.036,Z 634.5,A -85,B 0,C 180,E1 -1890,E2 -1890} C_VEL
LIN {X 0,Y 580.041,Z 633.83,A -85,B 0,C 180,E1 -1891.389,E2 -1891.389} C_VEL
LIN {X 0,Y 580.041,Z 631.835,A -85,B 0,C 180,E1 -1892.778,E2 -1892.778} C_VEL
LIN {X 0,Y 580.102,Z 628.447,A -85,B 0,C 180,E1 -1894.169,E2 -1894.169} C_VEL
LIN {X 0,Y 580.128,Z 623.574,A -85,B 0,C 180,E1 -1895.562,E2 -1895.562} C_VEL
LIN {X 0,Y 580.141,Z 617.058,A -85,B 0,C 180,E1 -1896.958,E2 -1896.958} C_VEL
LIN {X 0,Y 580.192,Z 609.803,A -85,B 0,C 180,E1 -1898.183,E2 -1898.183} C_VEL
LIN {X 0,Y 580.284,Z 600.824,A -85,B 0,C 180,E1 -1899.41,E2 -1899.41} C_VEL
LIN {X 0,Y 580.356,Z 591.391,A -85,B 0,C 180,E1 -1900.466,E2 -1900.466} C_VEL
LIN {X 0,Y 580.475,Z 581.312,A -85,B 0,C 180,E1 -1901.404,E2 -1901.404} C_VEL
LIN {X 0,Y 580.592,Z 569.428,A -85,B 0,C 180,E1 -1902.319,E2 -1902.319} C_VEL
LIN {X 0,Y 580.715,Z 556.652,A -85,B 0,C 180,E1 -1903.116,E2 -1903.116} C_VEL
LIN {X 0,Y 580.894,Z 543.188,A -85,B 0,C 180,E1 -1903.78,E2 -1903.78} C_VEL
LIN {X 0,Y 581.02,Z 529.509,A -85,B 0,C 180,E1 -1904.293,E2 -1904.293} C_VEL
LIN {X 0,Y 581.104,Z 515.516,A -85,B 0,C 180,E1 -1904.67,E2 -1904.67} C_VEL
LIN {X 0,Y 580.958,Z 506.573,A -85,B 0,C 180,E1 -1904.838,E2 -1904.838} C_VEL
LIN {X 0,Y 580.175,Z 502.42,A -85,B 0,C 180,E1 -1904.939,E2 -1904.939} C_VEL
LIN {X 0,Y 580.227,Z 493.319,A -85,B 0,C 180,E1 -1907.627,E2 -1907.627} C_VEL
LIN {X 0,Y 580.271,Z 484.752,A -85,B 0,C 180,E1 -1910.193,E2 -1910.193} C_VEL
LIN {X 0,Y 580.312,Z 476.186,A -85,B 0,C 180,E1 -1912.802,E2 -1912.802} C_VEL
LIN {X 0,Y 580.393,Z 467.62,A -85,B 0,C 180,E1 -1915.459,E2 -1915.459} C_VEL
LIN {X 0,Y 580.506,Z 457.83,A -85,B 0,C 180,E1 -1918.569,E2 -1918.569} C_VEL
LIN {X 0,Y 580.541,Z 449.264,A -85,B 0,C 180,E1 -1921.37,E2 -1921.37} C_VEL
LIN {X 0,Y 580.67,Z 440.777,A -85,B 0,C 180,E1 -1924.223,E2 -1924.223} C_VEL
LIN {X 0,Y 580.747,Z 432.131,A -85,B 0,C 180,E1 -1927.235,E2 -1927.235} C_VEL
LIN {X 0,Y 580.707,Z 424.115,A -85,B 0,C 180,E1 -1929.899,E2 -1929.899} C_VEL
LIN {X 0,Y 580.712,Z 415.012,A -85,B 0,C 180,E1 -1933.051,E2 -1933.051} C_VEL
LIN {X 0,Y 580.847,Z 406.927,A -85,B 0,C 180,E1 -1935.98,E2 -1935.98} C_VEL
LIN {X 0,Y 580.315,Z 401.826,A -85,B 0,C 180,E1 -1937.957,E2 -1937.957} C_VEL
LIN {X 0,Y 580.276,Z 401.833,A -85,B 0,C 180,E1 -1940.965,E2 -1940.965} C_VEL
LIN {X 0,Y 580.283,Z 401.829,A -85,B 0,C 180,E1 -1943.597,E2 -1943.597} C_VEL
LIN {X 0,Y 580.319,Z 401.822,A -85,B 0,C 180,E1 -1946.145,E2 -1946.145} C_VEL
LIN {X 0,Y 580.28,Z 401.83,A -85,B 0,C 180,E1 -1948.615,E2 -1948.615} C_VEL
LIN {X 0,Y 580.296,Z 401.826,A -85,B 0,C 180,E1 -1951.024,E2 -1951.024} C_VEL
LIN {X 0,Y 580.295,Z 401.823,A -85,B 0,C 180,E1 -1953.666,E2 -1953.666} C_VEL
LIN {X 0,Y 580.304,Z 401.826,A -85,B 0,C 180,E1 -1955.684,E2 -1955.684} C_VEL
LIN {X 0,Y 580.276,Z 401.827,A -85,B 0,C 180,E1 -1957.948,E2 -1957.948} C_VEL
LIN {X 0,Y 580.303,Z 401.824,A -85,B 0,C 180,E1 -1960.914,E2 -1960.914} C_VEL
LIN {X 0,Y 580.334,Z 401.822,A -85,B 0,C 180,E1 -1963.103,E2 -1963.103} C_VEL
LIN {X 0,Y 580.327,Z 401.82,A -85,B 0,C 180,E1 -1965.983,E2 -1965.983} C_VEL
LIN {X 0,Y 580.308,Z 401.823,A -85,B 0,C 180,E1 -1968.827,E2 -1968.827} C_VEL
LIN {X 0,Y 580.314,Z 401.821,A -85,B 0,C 180,E1 -1971.644,E2 -1971.644} C_VEL
LIN {X 0,Y 580.291,Z 401.828,A -85,B 0,C 180,E1 -1973.742,E2 -1973.742} C_VEL
LIN {X 0,Y 580.267,Z 401.829,A -85,B 0,C 180,E1 -1975.833,E2 -1975.833} C_VEL
LIN {X 0,Y 580.334,Z 401.819,A -85,B 0,C 180,E1 -1977.918,E2 -1977.918} C_VEL
LIN {X 0,Y 580.363,Z 401.816,A -85,B 0,C 180,E1 -1980.694,E2 -1980.694} C_VEL
LIN {X 0,Y 580.282,Z 401.826,A -85,B 0,C 180,E1 -1983.472,E2 -1983.472} C_VEL
LIN {X 0,Y 580.324,Z 401.822,A -85,B 0,C 180,E1 -1985.56,E2 -1985.56} C_VEL
LIN {X 0,Y 580.335,Z 401.818,A -85,B 0,C 180,E1 -1988.356,E2 -1988.356} C_VEL
LIN {X 0,Y 580.303,Z 401.824,A -85,B 0,C 180,E1 -1991.191,E2 -1991.191} C_VEL
LIN {X 0,Y 580.327,Z 401.82,A -85,B 0,C 180,E1 -1994.017,E2 -1994.017} C_VEL
LIN {X 0,Y 580.315,Z 401.824,A -85,B 0,C 180,E1 -1996.914,E2 -1996.914} C_VEL
LIN {X 0,Y 580.308,Z 401.826,A -85,B 0,C 180,E1 -1999.822,E2 -1999.822} C_VEL
LIN {X 0,Y 580.286,Z 401.828,A -85,B 0,C 180,E1 -2001.333,E2 -2001.333} C_VEL
LIN {X 0,Y 579.589,Z 401.913,A -85,B 0,C 180,E1 -2001.912,E2 -2001.912} C_VEL
LIN {X 0,Y 576.711,Z 402.273,A -85,B 0,C 180,E1 -2002.852,E2 -2002.852} C_VEL
LIN {X 0,Y 574.316,Z 402.57,A -85,B 0,C 180,E1 -2003.608,E2 -2003.608} C_VEL
LIN {X 0,Y 573.318,Z 402.698,A -85,B 0,C 180,E1 -2004.192,E2 -2004.192} C_VEL
LIN {X 0,Y 573.252,Z 402.702,A -85,B 0,C 180,E1 -2004.389,E2 -2004.389} C_VEL
LIN {X 0,Y 573.255,Z 402.705,A -85,B 0,C 180,E1 -2006.976,E2 -2006.976} C_VEL
LIN {X 0,Y 573.249,Z 402.702,A -85,B 0,C 180,E1 -2009.488,E2 -2009.488} C_VEL
LIN {X 0,Y 573.258,Z 402.702,A -85,B 0,C 180,E1 -2012.645,E2 -2012.645} C_VEL
LIN {X 0,Y 573.208,Z 402.707,A -85,B 0,C 180,E1 -2015.188,E2 -2015.188} C_VEL
LIN {X 0,Y 573.239,Z 402.707,A -85,B 0,C 180,E1 -2017.807,E2 -2017.807} C_VEL
LIN {X 0,Y 573.247,Z 402.707,A -85,B 0,C 180,E1 -2020.525,E2 -2020.525} C_VEL
LIN {X 0,Y 573.25,Z 402.705,A -85,B 0,C 180,E1 -2023.358,E2 -2023.358} C_VEL
LIN {X 0,Y 573.246,Z 402.706,A -85,B 0,C 180,E1 -2026.331,E2 -2026.331} C_VEL
LIN {X 0,Y 573.262,Z 402.707,A -85,B 0,C 180,E1 -2029.476,E2 -2029.476} C_VEL
LIN {X 0,Y 573.301,Z 402.782,A -85,B 0,C 180,E1 -2031.522,E2 -2031.522} C_VEL
LIN {X 0,Y 573.661,Z 407.745,A -85,B 0,C 180,E1 -2032.781,E2 -2032.781} C_VEL
LIN {X 0,Y 573.509,Z 418.878,A -85,B 0,C 180,E1 -2035.688,E2 -2035.688} C_VEL
LIN {X 0,Y 573.564,Z 428.407,A -85,B 0,C 180,E1 -2038.205,E2 -2038.205} C_VEL
LIN {X 0,Y 573.594,Z 439.289,A -85,B 0,C 180,E1 -2041.055,E2 -2041.055} C_VEL
LIN {X 0,Y 573.555,Z 448.26,A -85,B 0,C 180,E1 -2043.444,E2 -2043.444} C_VEL
LIN {X 0,Y 573.431,Z 458.158,A -85,B 0,C 180,E1 -2046.143,E2 -2046.143} C_VEL
LIN {X 0,Y 573.364,Z 467.644,A -85,B 0,C 180,E1 -2048.681,E2 -2048.681} C_VEL
LIN {X 0,Y 573.244,Z 478.039,A -85,B 0,C 180,E1 -2051.412,E2 -2051.412} C_VEL
LIN {X 0,Y 573.178,Z 487.981,A -85,B 0,C 180,E1 -2053.985,E2 -2053.985} C_VEL
LIN {X 0,Y 573.171,Z 491.75,A -85,B 0,C 180,E1 -2054.931,E2 -2054.931} C_VEL
LIN {X 0,Y 574.288,Z 498.56,A -85,B 0,C 180,E1 -2055.063,E2 -2055.063} C_VEL
LIN {X 0,Y 574.166,Z 513.136,A -85,B 0,C 180,E1 -2055.386,E2 -2055.386} C_VEL
LIN {X 0,Y 574.014,Z 527.749,A -85,B 0,C 180,E1 -2055.871,E2 -2055.871} C_VEL
LIN {X 0,Y 573.903,Z 540.783,A -85,B 0,C 180,E1 -2056.455,E2 -2056.455} C_VEL
LIN {X 0,Y 573.713,Z 553.402,A -85,B 0,C 180,E1 -2057.172,E2 -2057.172} C_VEL
LIN {X 0,Y 573.535,Z 566.071,A -85,B 0,C 180,E1 -2058.066,E2 -2058.066} C_VEL
LIN {X 0,Y 573.438,Z 577.711,A -85,B 0,C 180,E1 -2059.081,E2 -2059.081} C_VEL
LIN {X 0,Y 573.245,Z 587.477,A -85,B 0,C 180,E1 -2060.117,E2 -2060.117} C_VEL
LIN {X 0,Y 573.202,Z 595.869,A -85,B 0,C 180,E1 -2061.184,E2 -2061.184} C_VEL
LIN {X 0,Y 573.111,Z 603.875,A -85,B 0,C 180,E1 -2062.425,E2 -2062.425} C_VEL
LIN {X 0,Y 573.022,Z 610.333,A -85,B 0,C 180,E1 -2063.663,E2 -2063.663} C_VEL
LIN {X 0,Y 573,Z 614.79,A -85,B 0,C 180,E1 -2064.722,E2 -2064.722} C_VEL
LIN {X 0,Y 573.029,Z 618.314,A -85,B 0,C 180,E1 -2065.78,E2 -2065.78} C_VEL
LIN {X 0,Y 572.957,Z 621.749,A -85,B 0,C 180,E1 -2067.188,E2 -2067.188} C_VEL
LIN {X 0,Y 572.944,Z 623.786,A -85,B 0,C 180,E1 -2068.594,E2 -2068.594} C_VEL
LIN {X 0,Y 572.937,Z 624.496,A -85,B 0,C 180,E1 -2070,E2 -2070} C_VEL
LIN {X 0,Y 572.941,Z 623.872,A -85,B 0,C 180,E1 -2071.406,E2 -2071.406} C_VEL
LIN {X 0,Y 572.954,Z 621.93,A -85,B 0,C 180,E1 -2072.812,E2 -2072.812} C_VEL
LIN {X 0,Y 573.03,Z 618.581,A -85,B 0,C 180,E1 -2074.22,E2 -2074.22} C_VEL
LIN {X 0,Y 573.057,Z 613.763,A -85,B 0,C 180,E1 -2075.63,E2 -2075.63} C_VEL
LIN {X 0,Y 573.054,Z 607.29,A -85,B 0,C 180,E1 -2077.045,E2 -2077.045} C_VEL
LIN {X 0,Y 573.143,Z 600.094,A -85,B 0,C 180,E1 -2078.284,E2 -2078.284} C_VEL
LIN {X 0,Y 573.225,Z 591.171,A -85,B 0,C 180,E1 -2079.527,E2 -2079.527} C_VEL
LIN {X 0,Y 573.351,Z 581.838,A -85,B 0,C 180,E1 -2080.595,E2 -2080.595} C_VEL
LIN {X 0,Y 573.476,Z 570.438,A -85,B 0,C 180,E1 -2081.666,E2 -2081.666} C_VEL
LIN {X 0,Y 573.642,Z 558.807,A -85,B 0,C 180,E1 -2082.56,E2 -2082.56} C_VEL
LIN {X 0,Y 573.812,Z 545.866,A -85,B 0,C 180,E1 -2083.367,E2 -2083.367} C_VEL
LIN {X 0,Y 573.994,Z 533.187,A -85,B 0,C 180,E1 -2083.994,E2 -2083.994} C_VEL
LIN {X 0,Y 574.129,Z 519.78,A -85,B 0,C 180,E1 -2084.503,E2 -2084.503} C_VEL
LIN {X 0,Y 574.278,Z 505.48,A -85,B 0,C 180,E1 -2084.892,E2 -2084.892} C_VEL
LIN {X 0,Y 574.048,Z 496.372,A -85,B 0,C 180,E1 -2085.07,E2 -2085.07} C_VEL
LIN {X 0,Y 573.181,Z 491.616,A -85,B 0,C 180,E1 -2085.171,E2 -2085.171} C_VEL
LIN {X 0,Y 573.242,Z 479.805,A -85,B 0,C 180,E1 -2088.218,E2 -2088.218} C_VEL
LIN {X 0,Y 573.311,Z 469.859,A -85,B 0,C 180,E1 -2090.824,E2 -2090.824} C_VEL
LIN {X 0,Y 573.385,Z 459.911,A -85,B 0,C 180,E1 -2093.476,E2 -2093.476} C_VEL
LIN {X 0,Y 573.553,Z 449.965,A -85,B 0,C 180,E1 -2096.176,E2 -2096.176} C_VEL
